Fanuc TP program (LS listing): ultrahose1.ls

/PROG  ultrahose1
/ATTR
COMMENT	= "19-03-19 19:07:18";
PROG_SIZE	= 0;
DEFAULT_GROUP	= 1, *, *, *, *;
/APPL
    ARC Welding Equipment: 1, *, *, *, *;
/MN
   1:  CALL HOME_ALL;
   1:  UFRAME_NUM = 1;
   1:  UTOOL_NUM = 3;
   1:  COL GUARD ADJUST 150;
   1:  PR[91] = PR[90];
   1:  PR[91,1] = PR[90,1] + 11.874;
   1:  PR[91,2] = PR[90,2] + -13.968;
   1:  PR[91,3] = PR[90,3] + 19.695;
   1:  PR[92] = PR[91];
   1:  PR[92,3] = PR[92,3] + 20;
   1:J PR[92] 10% FINE;
   1:L PR[91] R[100]mm/sec CNT100;
   1:  CALL LASER_DRAHT_START;
   1:  PR[91,1] = PR[90,1] + 15.068;
   1:  PR[91,2] = PR[90,2] + -16.411;
   1:L PR[91] R[100]mm/sec CNT100;
   1:  PR[91,1] = PR[90,1] + 15.529;
   1:  PR[91,2] = PR[90,2] + -16.733;
   1:L PR[91] R[100]mm/sec CNT100;
   1:  PR[91,1] = PR[90,1] + 16.034;
   1:  PR[91,2] = PR[90,2] + -16.968;
   1:L PR[91] R[100]mm/sec CNT100;
   1:  PR[91,1] = PR[90,1] + 19.725;
   1:  PR[91,2] = PR[90,2] + -18.490;
   1:L PR[91] R[100]mm/sec CNT100;
   1:  PR[91,1] = PR[90,1] + 20.251;
   1:  PR[91,2] = PR[90,2] + -18.631;
   1:L PR[91] R[100]mm/sec CNT100;
   1:  PR[91,1] = PR[90,1] + 24.153;
   1:  PR[91,2] = PR[90,2] + -19.139;
   1:L PR[91] R[100]mm/sec CNT100;
   1:  PR[91,1] = PR[90,1] + 24.768;
   1:  PR[91,2] = PR[90,2] + -19.192;
   1:L PR[91] R[100]mm/sec CNT100;
   1:  PR[91,1] = PR[90,1] + 25.380;
   1:  PR[91,2] = PR[90,2] + -19.139;
   1:L PR[91] R[100]mm/sec CNT100;
   1:  PR[91,1] = PR[90,1] + 29.249;
   1:  PR[91,2] = PR[90,2] + -18.622;
   1:L PR[91] R[100]mm/sec CNT100;
   1:  PR[91,1] = PR[90,1] + 29.789;
   1:  PR[91,2] = PR[90,2] + -18.477;
   1:L PR[91] R[100]mm/sec CNT100;
   1:  PR[91,1] = PR[90,1] + 30.450;
   1:  PR[91,2] = PR[90,2] + -18.169;
   1:L PR[91] R[100]mm/sec CNT100;
   1:  PR[91,1] = PR[90,1] + 34.024;
   1:  PR[91,2] = PR[90,2] + -16.681;
   1:L PR[91] R[100]mm/sec CNT100;
   1:  PR[91,1] = PR[90,1] + 34.539;
   1:  PR[91,2] = PR[90,2] + -16.320;
   1:L PR[91] R[100]mm/sec CNT100;
   1:  PR[91,1] = PR[90,1] + 37.568;
   1:  PR[91,2] = PR[90,2] + -13.991;
   1:L PR[91] R[100]mm/sec CNT100;
   1:  PR[91,1] = PR[90,1] + 38.026;
   1:  PR[91,2] = PR[90,2] + -13.533;
   1:L PR[91] R[100]mm/sec CNT100;
   1:  PR[91,1] = PR[90,1] + 40.324;
   1:  PR[91,2] = PR[90,2] + -10.530;
   1:L PR[91] R[100]mm/sec CNT100;
   1:  PR[91,1] = PR[90,1] + 40.733;
   1:  PR[91,2] = PR[90,2] + -9.947;
   1:L PR[91] R[100]mm/sec CNT100;
   1:  PR[91,1] = PR[90,1] + 41.032;
   1:  PR[91,2] = PR[90,2] + -9.305;
   1:L PR[91] R[100]mm/sec CNT100;
   1:  PR[91,1] = PR[90,1] + 42.471;
   1:  PR[91,2] = PR[90,2] + -5.824;
   1:L PR[91] R[100]mm/sec CNT100;
   1:  PR[91,1] = PR[90,1] + 42.635;
   1:  PR[91,2] = PR[90,2] + -5.212;
   1:L PR[91] R[100]mm/sec CNT100;
   1:  PR[91,1] = PR[90,1] + 42.704;
   1:  PR[91,2] = PR[90,2] + -4.424;
   1:L PR[91] R[100]mm/sec CNT100;
   1:  PR[91,1] = PR[90,1] + 43.146;
   1:  PR[91,2] = PR[90,2] + -0.638;
   1:L PR[91] R[100]mm/sec CNT100;
   1:  PR[91,1] = PR[90,1] + 43.128;
   1:  PR[91,2] = PR[90,2] + 0.046;
   1:L PR[91] R[100]mm/sec CNT100;
   1:  PR[91,1] = PR[90,1] + 42.647;
   1:  PR[91,2] = PR[90,2] + 3.711;
   1:L PR[91] R[100]mm/sec CNT100;
   1:  PR[91,1] = PR[90,1] + 42.471;
   1:  PR[91,2] = PR[90,2] + 4.366;
   1:L PR[91] R[100]mm/sec CNT100;
   1:  PR[91,1] = PR[90,1] + 41.032;
   1:  PR[91,2] = PR[90,2] + 7.846;
   1:L PR[91] R[100]mm/sec CNT100;
   1:  PR[91,1] = PR[90,1] + 40.733;
   1:  PR[91,2] = PR[90,2] + 8.488;
   1:L PR[91] R[100]mm/sec CNT100;
   1:  PR[91,1] = PR[90,1] + 40.324;
   1:  PR[91,2] = PR[90,2] + 9.072;
   1:L PR[91] R[100]mm/sec CNT100;
   1:  PR[91,1] = PR[90,1] + 38.025;
   1:  PR[91,2] = PR[90,2] + 12.075;
   1:L PR[91] R[100]mm/sec CNT100;
   1:  PR[91,1] = PR[90,1] + 37.567;
   1:  PR[91,2] = PR[90,2] + 12.533;
   1:L PR[91] R[100]mm/sec CNT100;
   1:  PR[91,1] = PR[90,1] + 34.538;
   1:  PR[91,2] = PR[90,2] + 14.862;
   1:L PR[91] R[100]mm/sec CNT100;
   1:  PR[91,1] = PR[90,1] + 33.989;
   1:  PR[91,2] = PR[90,2] + 15.247;
   1:L PR[91] R[100]mm/sec CNT100;
   1:  PR[91,1] = PR[90,1] + 33.379;
   1:  PR[91,2] = PR[90,2] + 15.531;
   1:L PR[91] R[100]mm/sec CNT100;
   1:  PR[91,1] = PR[90,1] + 29.828;
   1:  PR[91,2] = PR[90,2] + 17.008;
   1:L PR[91] R[100]mm/sec CNT100;
   1:  PR[91,1] = PR[90,1] + 29.246;
   1:  PR[91,2] = PR[90,2] + 17.164;
   1:L PR[91] R[100]mm/sec CNT100;
   1:  PR[91,1] = PR[90,1] + 25.377;
   1:  PR[91,2] = PR[90,2] + 17.680;
   1:L PR[91] R[100]mm/sec CNT100;
   1:  PR[91,1] = PR[90,1] + 24.766;
   1:  PR[91,2] = PR[90,2] + 17.734;
   1:L PR[91] R[100]mm/sec CNT100;
   1:  PR[91,1] = PR[90,1] + 24.150;
   1:  PR[91,2] = PR[90,2] + 17.680;
   1:L PR[91] R[100]mm/sec CNT100;
   1:  PR[91,1] = PR[90,1] + 20.249;
   1:  PR[91,2] = PR[90,2] + 17.172;
   1:L PR[91] R[100]mm/sec CNT100;
   1:  PR[91,1] = PR[90,1] + 19.767;
   1:  PR[91,2] = PR[90,2] + 17.043;
   1:L PR[91] R[100]mm/sec CNT100;
   1:  PR[91,1] = PR[90,1] + 19.155;
   1:  PR[91,2] = PR[90,2] + 16.757;
   1:L PR[91] R[100]mm/sec CNT100;
   1:  PR[91,1] = PR[90,1] + 15.490;
   1:  PR[91,2] = PR[90,2] + 15.247;
   1:L PR[91] R[100]mm/sec CNT100;
   1:  PR[91,1] = PR[90,1] + 15.067;
   1:  PR[91,2] = PR[90,2] + 14.951;
   1:L PR[91] R[100]mm/sec CNT100;
   1:  PR[91,1] = PR[90,1] + 11.873;
   1:  PR[91,2] = PR[90,2] + 12.508;
   1:L PR[91] R[100]mm/sec CNT100;
   1:  PR[91,1] = PR[90,1] + 11.527;
   1:  PR[91,2] = PR[90,2] + 12.162;
   1:L PR[91] R[100]mm/sec CNT100;
   1:  PR[91,1] = PR[90,1] + 9.049;
   1:  PR[91,2] = PR[90,2] + 8.939;
   1:L PR[91] R[100]mm/sec CNT100;
   1:  PR[91,1] = PR[90,1] + 8.753;
   1:  PR[91,2] = PR[90,2] + 8.515;
   1:L PR[91] R[100]mm/sec CNT100;
   1:  PR[91,1] = PR[90,1] + 8.534;
   1:  PR[91,2] = PR[90,2] + 8.047;
   1:L PR[91] R[100]mm/sec CNT100;
   1:  PR[91,1] = PR[90,1] + 6.970;
   1:  PR[91,2] = PR[90,2] + 4.277;
   1:L PR[91] R[100]mm/sec CNT100;
   1:  PR[91,1] = PR[90,1] + 6.862;
   1:  PR[91,2] = PR[90,2] + 3.874;
   1:L PR[91] R[100]mm/sec CNT100;
   1:  PR[91,1] = PR[90,1] + 6.811;
   1:  PR[91,2] = PR[90,2] + 3.287;
   1:L PR[91] R[100]mm/sec CNT100;
   1:  PR[91,1] = PR[90,1] + 6.282;
   1:  PR[91,2] = PR[90,2] + -0.772;
   1:L PR[91] R[100]mm/sec CNT100;
   1:  PR[91,1] = PR[90,1] + 6.336;
   1:  PR[91,2] = PR[90,2] + -1.394;
   1:L PR[91] R[100]mm/sec CNT100;
   1:  PR[91,1] = PR[90,1] + 6.851;
   1:  PR[91,2] = PR[90,2] + -5.290;
   1:L PR[91] R[100]mm/sec CNT100;
   1:  PR[91,1] = PR[90,1] + 6.970;
   1:  PR[91,2] = PR[90,2] + -5.736;
   1:L PR[91] R[100]mm/sec CNT100;
   1:  PR[91,1] = PR[90,1] + 8.535;
   1:  PR[91,2] = PR[90,2] + -9.506;
   1:L PR[91] R[100]mm/sec CNT100;
   1:  PR[91,1] = PR[90,1] + 8.753;
   1:  PR[91,2] = PR[90,2] + -9.975;
   1:L PR[91] R[100]mm/sec CNT100;
   1:  PR[91,1] = PR[90,1] + 9.050;
   1:  PR[91,2] = PR[90,2] + -10.398;
   1:L PR[91] R[100]mm/sec CNT100;
   1:  PR[91,1] = PR[90,1] + 11.528;
   1:  PR[91,2] = PR[90,2] + -13.622;
   1:L PR[91] R[100]mm/sec CNT100;
   1:  PR[91,1] = PR[90,1] + 11.874;
   1:  PR[91,2] = PR[90,2] + -13.968;
   1:L PR[91] R[100]mm/sec CNT100TB   .50sec,CALL END_PUD;
   1:  PR[92] = PR[91];
   1:  PR[92,3] = PR[92,3] + 20;
   1:J PR[92] 10% FINE;
   1:  PR[91,1] = PR[90,1] + 59.086;
   1:  PR[91,2] = PR[90,2] + -12.393;
   1:  PR[92] = PR[91];
   1:  PR[92,3] = PR[92,3] + 20;
   1:J PR[92] 10% FINE;
   1:L PR[91] R[100]mm/sec CNT100;
   1:  CALL LASER_DRAHT_START;
   1:  PR[91,1] = PR[90,1] + 60.293;
   1:  PR[91,2] = PR[90,2] + -13.557;
   1:L PR[91] R[100]mm/sec CNT100;
   1:  PR[91,1] = PR[90,1] + 62.143;
   1:  PR[91,2] = PR[90,2] + -15.300;
   1:L PR[91] R[100]mm/sec CNT100;
   1:  PR[91,1] = PR[90,1] + 63.971;
   1:  PR[91,2] = PR[90,2] + -16.401;
   1:L PR[91] R[100]mm/sec CNT100;
   1:  PR[91,1] = PR[90,1] + 65.772;
   1:  PR[91,2] = PR[90,2] + -17.456;
   1:L PR[91] R[100]mm/sec CNT100;
   1:  PR[91,1] = PR[90,1] + 68.248;
   1:  PR[91,2] = PR[90,2] + -18.274;
   1:L PR[91] R[100]mm/sec CNT100;
   1:  PR[91,1] = PR[90,1] + 69.782;
   1:  PR[91,2] = PR[90,2] + -18.759;
   1:L PR[91] R[100]mm/sec CNT100;
   1:  PR[91,1] = PR[90,1] + 72.825;
   1:  PR[91,2] = PR[90,2] + -19.060;
   1:L PR[91] R[100]mm/sec CNT100;
   1:  PR[91,1] = PR[90,1] + 73.969;
   1:  PR[91,2] = PR[90,2] + -19.158;
   1:L PR[91] R[100]mm/sec CNT100;
   1:  PR[91,1] = PR[90,1] + 78.141;
   1:  PR[91,2] = PR[90,2] + -18.634;
   1:L PR[91] R[100]mm/sec CNT100;
   1:  PR[91,1] = PR[90,1] + 81.686;
   1:  PR[91,2] = PR[90,2] + -17.372;
   1:L PR[91] R[100]mm/sec CNT100;
   1:  PR[91,1] = PR[90,1] + 82.061;
   1:  PR[91,2] = PR[90,2] + -17.234;
   1:L PR[91] R[100]mm/sec CNT100;
   1:  PR[91,1] = PR[90,1] + 85.575;
   1:  PR[91,2] = PR[90,2] + -15.011;
   1:L PR[91] R[100]mm/sec CNT100;
   1:  PR[91,1] = PR[90,1] + 88.491;
   1:  PR[91,2] = PR[90,2] + -12.096;
   1:L PR[91] R[100]mm/sec CNT100;
   1:  PR[91,1] = PR[90,1] + 90.677;
   1:  PR[91,2] = PR[90,2] + -8.631;
   1:L PR[91] R[100]mm/sec CNT100;
   1:  PR[91,1] = PR[90,1] + 92.020;
   1:  PR[91,2] = PR[90,2] + -4.770;
   1:L PR[91] R[100]mm/sec CNT100;
   1:  PR[91,1] = PR[90,1] + 92.467;
   1:  PR[91,2] = PR[90,2] + -0.729;
   1:L PR[91] R[100]mm/sec CNT100;
   1:  PR[91,1] = PR[90,1] + 92.020;
   1:  PR[91,2] = PR[90,2] + 3.311;
   1:L PR[91] R[100]mm/sec CNT100;
   1:  PR[91,1] = PR[90,1] + 90.677;
   1:  PR[91,2] = PR[90,2] + 7.172;
   1:L PR[91] R[100]mm/sec CNT100;
   1:  PR[91,1] = PR[90,1] + 88.491;
   1:  PR[91,2] = PR[90,2] + 10.637;
   1:L PR[91] R[100]mm/sec CNT100;
   1:  PR[91,1] = PR[90,1] + 85.575;
   1:  PR[91,2] = PR[90,2] + 13.552;
   1:L PR[91] R[100]mm/sec CNT100;
   1:  PR[91,1] = PR[90,1] + 82.069;
   1:  PR[91,2] = PR[90,2] + 15.770;
   1:L PR[91] R[100]mm/sec CNT100;
   1:  PR[91,1] = PR[90,1] + 78.143;
   1:  PR[91,2] = PR[90,2] + 17.175;
   1:L PR[91] R[100]mm/sec CNT100;
   1:  PR[91,1] = PR[90,1] + 74.809;
   1:  PR[91,2] = PR[90,2] + 17.581;
   1:L PR[91] R[100]mm/sec CNT100;
   1:  PR[91,1] = PR[90,1] + 73.972;
   1:  PR[91,2] = PR[90,2] + 17.696;
   1:L PR[91] R[100]mm/sec CNT100;
   1:  PR[91,1] = PR[90,1] + 70.968;
   1:  PR[91,2] = PR[90,2] + 17.396;
   1:L PR[91] R[100]mm/sec CNT100;
   1:  PR[91,1] = PR[90,1] + 69.783;
   1:  PR[91,2] = PR[90,2] + 17.297;
   1:L PR[91] R[100]mm/sec CNT100;
   1:  PR[91,1] = PR[90,1] + 67.265;
   1:  PR[91,2] = PR[90,2] + 16.462;
   1:L PR[91] R[100]mm/sec CNT100;
   1:  PR[91,1] = PR[90,1] + 65.772;
   1:  PR[91,2] = PR[90,2] + 15.993;
   1:L PR[91] R[100]mm/sec CNT100;
   1:  PR[91,1] = PR[90,1] + 63.838;
   1:  PR[91,2] = PR[90,2] + 14.826;
   1:L PR[91] R[100]mm/sec CNT100;
   1:  PR[91,1] = PR[90,1] + 62.143;
   1:  PR[91,2] = PR[90,2] + 13.837;
   1:L PR[91] R[100]mm/sec CNT100;
   1:  PR[91,1] = PR[90,1] + 60.804;
   1:  PR[91,2] = PR[90,2] + 12.545;
   1:L PR[91] R[100]mm/sec CNT100;
   1:  PR[91,1] = PR[90,1] + 59.084;
   1:  PR[91,2] = PR[90,2] + 10.928;
   1:L PR[91] R[100]mm/sec CNT100;
   1:  PR[91,1] = PR[90,1] + 58.273;
   1:  PR[91,2] = PR[90,2] + 9.680;
   1:L PR[91] R[100]mm/sec CNT100;
   1:  PR[91,1] = PR[90,1] + 56.759;
   1:  PR[91,2] = PR[90,2] + 7.403;
   1:L PR[91] R[100]mm/sec CNT100;
   1:  PR[91,1] = PR[90,1] + 55.312;
   1:  PR[91,2] = PR[90,2] + 3.452;
   1:L PR[91] R[100]mm/sec CNT100;
   1:  PR[91,1] = PR[90,1] + 55.212;
   1:  PR[91,2] = PR[90,2] + 2.599;
   1:L PR[91] R[100]mm/sec CNT100;
   1:  PR[91,1] = PR[90,1] + 55.211;
   1:  PR[91,2] = PR[90,2] + 2.366;
   1:L PR[91] R[100]mm/sec CNT100;
   1:  PR[91,1] = PR[90,1] + 54.847;
   1:  PR[91,2] = PR[90,2] + -0.750;
   1:L PR[91] R[100]mm/sec CNT100;
   1:  PR[91,1] = PR[90,1] + 54.928;
   1:  PR[91,2] = PR[90,2] + -1.594;
   1:L PR[91] R[100]mm/sec CNT100;
   1:  PR[91,1] = PR[90,1] + 55.312;
   1:  PR[91,2] = PR[90,2] + -4.913;
   1:L PR[91] R[100]mm/sec CNT100;
   1:  PR[91,1] = PR[90,1] + 56.761;
   1:  PR[91,2] = PR[90,2] + -8.866;
   1:L PR[91] R[100]mm/sec CNT100;
   1:  PR[91,1] = PR[90,1] + 59.086;
   1:  PR[91,2] = PR[90,2] + -12.393;
   1:L PR[91] R[100]mm/sec CNT100TB   .50sec,CALL END_PUD;
   1:  PR[92] = PR[91];
   1:  PR[92,3] = PR[92,3] + 20;
   1:J PR[92] 10% FINE;
   1:  PR[91,1] = PR[90,1] + -40.837;
   1:  PR[91,2] = PR[90,2] + 7.347;
   1:  PR[92] = PR[91];
   1:  PR[92,3] = PR[92,3] + 20;
   1:J PR[92] 10% FINE;
   1:L PR[91] R[100]mm/sec CNT100;
   1:  CALL LASER_DRAHT_START;
   1:  PR[91,1] = PR[90,1] + -41.039;
   1:  PR[91,2] = PR[90,2] + 6.912;
   1:L PR[91] R[100]mm/sec CNT100;
   1:  PR[91,1] = PR[90,1] + -42.167;
   1:  PR[91,2] = PR[90,2] + 3.679;
   1:L PR[91] R[100]mm/sec CNT100;
   1:  PR[91,1] = PR[90,1] + -42.292;
   1:  PR[91,2] = PR[90,2] + 3.211;
   1:L PR[91] R[100]mm/sec CNT100;
   1:  PR[91,1] = PR[90,1] + -42.343;
   1:  PR[91,2] = PR[90,2] + 2.632;
   1:L PR[91] R[100]mm/sec CNT100;
   1:  PR[91,1] = PR[90,1] + -42.723;
   1:  PR[91,2] = PR[90,2] + -0.754;
   1:L PR[91] R[100]mm/sec CNT100;
   1:  PR[91,1] = PR[90,1] + -42.678;
   1:  PR[91,2] = PR[90,2] + -1.274;
   1:L PR[91] R[100]mm/sec CNT100;
   1:  PR[91,1] = PR[90,1] + -42.298;
   1:  PR[91,2] = PR[90,2] + -4.646;
   1:L PR[91] R[100]mm/sec CNT100;
   1:  PR[91,1] = PR[90,1] + -42.167;
   1:  PR[91,2] = PR[90,2] + -5.137;
   1:L PR[91] R[100]mm/sec CNT100;
   1:  PR[91,1] = PR[90,1] + -41.039;
   1:  PR[91,2] = PR[90,2] + -8.371;
   1:L PR[91] R[100]mm/sec CNT100;
   1:  PR[91,1] = PR[90,1] + -40.837;
   1:  PR[91,2] = PR[90,2] + -8.806;
   1:L PR[91] R[100]mm/sec CNT100;
   1:  PR[91,1] = PR[90,1] + -38.985;
   1:  PR[91,2] = PR[90,2] + -11.762;
   1:L PR[91] R[100]mm/sec CNT100;
   1:  PR[91,1] = PR[90,1] + -38.737;
   1:  PR[91,2] = PR[90,2] + -12.115;
   1:L PR[91] R[100]mm/sec CNT100;
   1:  PR[91,1] = PR[90,1] + -35.914;
   1:  PR[91,2] = PR[90,2] + -14.949;
   1:L PR[91] R[100]mm/sec CNT100;
   1:  PR[91,1] = PR[90,1] + -35.616;
   1:  PR[91,2] = PR[90,2] + -15.158;
   1:L PR[91] R[100]mm/sec CNT100;
   1:  PR[91,1] = PR[90,1] + -32.543;
   1:  PR[91,2] = PR[90,2] + -17.099;
   1:L PR[91] R[100]mm/sec CNT100;
   1:  PR[91,1] = PR[90,1] + -32.290;
   1:  PR[91,2] = PR[90,2] + -17.218;
   1:L PR[91] R[100]mm/sec CNT100;
   1:  PR[91,1] = PR[90,1] + -28.724;
   1:  PR[91,2] = PR[90,2] + -18.475;
   1:L PR[91] R[100]mm/sec CNT100;
   1:  PR[91,1] = PR[90,1] + -28.577;
   1:  PR[91,2] = PR[90,2] + -18.514;
   1:L PR[91] R[100]mm/sec CNT100;
   1:  PR[91,1] = PR[90,1] + -28.319;
   1:  PR[91,2] = PR[90,2] + -18.537;
   1:L PR[91] R[100]mm/sec CNT100;
   1:  PR[91,1] = PR[90,1] + -24.525;
   1:  PR[91,2] = PR[90,2] + -18.980;
   1:L PR[91] R[100]mm/sec CNT100;
   1:  PR[91,1] = PR[90,1] + -20.455;
   1:  PR[91,2] = PR[90,2] + -18.540;
   1:L PR[91] R[100]mm/sec CNT100;
   1:  PR[91,1] = PR[90,1] + -16.577;
   1:  PR[91,2] = PR[90,2] + -17.192;
   1:L PR[91] R[100]mm/sec CNT100;
   1:  PR[91,1] = PR[90,1] + -15.160;
   1:  PR[91,2] = PR[90,2] + -16.307;
   1:L PR[91] R[100]mm/sec CNT100;
   1:  PR[91,1] = PR[90,1] + -13.076;
   1:  PR[91,2] = PR[90,2] + -15.031;
   1:L PR[91] R[100]mm/sec CNT100;
   1:  PR[91,1] = PR[90,1] + -10.125;
   1:  PR[91,2] = PR[90,2] + -12.150;
   1:L PR[91] R[100]mm/sec CNT100;
   1:  PR[91,1] = PR[90,1] + -7.899;
   1:  PR[91,2] = PR[90,2] + -8.685;
   1:L PR[91] R[100]mm/sec CNT100;
   1:  PR[91,1] = PR[90,1] + -6.516;
   1:  PR[91,2] = PR[90,2] + -4.813;
   1:L PR[91] R[100]mm/sec CNT100;
   1:  PR[91,1] = PR[90,1] + -6.050;
   1:  PR[91,2] = PR[90,2] + -0.729;
   1:L PR[91] R[100]mm/sec CNT100;
   1:  PR[91,1] = PR[90,1] + -6.492;
   1:  PR[91,2] = PR[90,2] + 3.146;
   1:L PR[91] R[100]mm/sec CNT100;
   1:  PR[91,1] = PR[90,1] + -6.516;
   1:  PR[91,2] = PR[90,2] + 3.353;
   1:L PR[91] R[100]mm/sec CNT100;
   1:  PR[91,1] = PR[90,1] + -7.899;
   1:  PR[91,2] = PR[90,2] + 7.226;
   1:L PR[91] R[100]mm/sec CNT100;
   1:  PR[91,1] = PR[90,1] + -10.125;
   1:  PR[91,2] = PR[90,2] + 10.691;
   1:L PR[91] R[100]mm/sec CNT100;
   1:  PR[91,1] = PR[90,1] + -13.076;
   1:  PR[91,2] = PR[90,2] + 13.573;
   1:L PR[91] R[100]mm/sec CNT100;
   1:  PR[91,1] = PR[90,1] + -15.160;
   1:  PR[91,2] = PR[90,2] + 14.848;
   1:L PR[91] R[100]mm/sec CNT100;
   1:  PR[91,1] = PR[90,1] + -16.577;
   1:  PR[91,2] = PR[90,2] + 15.733;
   1:L PR[91] R[100]mm/sec CNT100;
   1:  PR[91,1] = PR[90,1] + -20.455;
   1:  PR[91,2] = PR[90,2] + 17.081;
   1:L PR[91] R[100]mm/sec CNT100;
   1:  PR[91,1] = PR[90,1] + -24.527;
   1:  PR[91,2] = PR[90,2] + 17.522;
   1:L PR[91] R[100]mm/sec CNT100;
   1:  PR[91,1] = PR[90,1] + -28.551;
   1:  PR[91,2] = PR[90,2] + 17.062;
   1:L PR[91] R[100]mm/sec CNT100;
   1:  PR[91,1] = PR[90,1] + -28.724;
   1:  PR[91,2] = PR[90,2] + 17.016;
   1:L PR[91] R[100]mm/sec CNT100;
   1:  PR[91,1] = PR[90,1] + -32.290;
   1:  PR[91,2] = PR[90,2] + 15.759;
   1:L PR[91] R[100]mm/sec CNT100;
   1:  PR[91,1] = PR[90,1] + -32.543;
   1:  PR[91,2] = PR[90,2] + 15.640;
   1:L PR[91] R[100]mm/sec CNT100;
   1:  PR[91,1] = PR[90,1] + -35.616;
   1:  PR[91,2] = PR[90,2] + 13.699;
   1:L PR[91] R[100]mm/sec CNT100;
   1:  PR[91,1] = PR[90,1] + -35.914;
   1:  PR[91,2] = PR[90,2] + 13.490;
   1:L PR[91] R[100]mm/sec CNT100;
   1:  PR[91,1] = PR[90,1] + -38.737;
   1:  PR[91,2] = PR[90,2] + 10.656;
   1:L PR[91] R[100]mm/sec CNT100;
   1:  PR[91,1] = PR[90,1] + -38.984;
   1:  PR[91,2] = PR[90,2] + 10.303;
   1:L PR[91] R[100]mm/sec CNT100;
   1:  PR[91,1] = PR[90,1] + -40.837;
   1:  PR[91,2] = PR[90,2] + 7.347;
   1:L PR[91] R[100]mm/sec CNT100TB   .50sec,CALL END_PUD;
   1:  PR[92] = PR[91];
   1:  PR[92,3] = PR[92,3] + 20;
   1:J PR[92] 10% FINE;
   1:  PR[91,1] = PR[90,1] + -83.415;
   1:  PR[91,2] = PR[90,2] + 14.998;
   1:  PR[92] = PR[91];
   1:  PR[92,3] = PR[92,3] + 20;
   1:J PR[92] 10% FINE;
   1:L PR[91] R[100]mm/sec CNT100;
   1:  CALL LASER_DRAHT_START;
   1:  PR[91,1] = PR[90,1] + -86.519;
   1:  PR[91,2] = PR[90,2] + 12.750;
   1:L PR[91] R[100]mm/sec CNT100;
   1:  PR[91,1] = PR[90,1] + -89.079;
   1:  PR[91,2] = PR[90,2] + 9.920;
   1:L PR[91] R[100]mm/sec CNT100;
   1:  PR[91,1] = PR[90,1] + -90.989;
   1:  PR[91,2] = PR[90,2] + 6.634;
   1:L PR[91] R[100]mm/sec CNT100;
   1:  PR[91,1] = PR[90,1] + -92.167;
   1:  PR[91,2] = PR[90,2] + 3.033;
   1:L PR[91] R[100]mm/sec CNT100;
   1:  PR[91,1] = PR[90,1] + -92.552;
   1:  PR[91,2] = PR[90,2] + -0.594;
   1:L PR[91] R[100]mm/sec CNT100;
   1:  PR[91,1] = PR[90,1] + -92.516;
   1:  PR[91,2] = PR[90,2] + -0.742;
   1:L PR[91] R[100]mm/sec CNT100;
   1:  PR[91,1] = PR[90,1] + -92.124;
   1:  PR[91,2] = PR[90,2] + -4.484;
   1:L PR[91] R[100]mm/sec CNT100;
   1:  PR[91,1] = PR[90,1] + -92.092;
   1:  PR[91,2] = PR[90,2] + -4.604;
   1:L PR[91] R[100]mm/sec CNT100;
   1:  PR[91,1] = PR[90,1] + -90.966;
   1:  PR[91,2] = PR[90,2] + -8.078;
   1:L PR[91] R[100]mm/sec CNT100;
   1:  PR[91,1] = PR[90,1] + -90.932;
   1:  PR[91,2] = PR[90,2] + -8.151;
   1:L PR[91] R[100]mm/sec CNT100;
   1:  PR[91,1] = PR[90,1] + -89.070;
   1:  PR[91,2] = PR[90,2] + -11.382;
   1:L PR[91] R[100]mm/sec CNT100;
   1:  PR[91,1] = PR[90,1] + -89.064;
   1:  PR[91,2] = PR[90,2] + -11.391;
   1:L PR[91] R[100]mm/sec CNT100;
   1:  PR[91,1] = PR[90,1] + -86.510;
   1:  PR[91,2] = PR[90,2] + -14.226;
   1:L PR[91] R[100]mm/sec CNT100;
   1:  PR[91,1] = PR[90,1] + -83.462;
   1:  PR[91,2] = PR[90,2] + -16.448;
   1:L PR[91] R[100]mm/sec CNT100;
   1:  PR[91,1] = PR[90,1] + -79.943;
   1:  PR[91,2] = PR[90,2] + -18.018;
   1:L PR[91] R[100]mm/sec CNT100;
   1:  PR[91,1] = PR[90,1] + -76.158;
   1:  PR[91,2] = PR[90,2] + -18.839;
   1:L PR[91] R[100]mm/sec CNT100;
   1:  PR[91,1] = PR[90,1] + -72.275;
   1:  PR[91,2] = PR[90,2] + -18.873;
   1:L PR[91] R[100]mm/sec CNT100;
   1:  PR[91,1] = PR[90,1] + -68.461;
   1:  PR[91,2] = PR[90,2] + -18.113;
   1:L PR[91] R[100]mm/sec CNT100;
   1:  PR[91,1] = PR[90,1] + -64.885;
   1:  PR[91,2] = PR[90,2] + -16.588;
   1:L PR[91] R[100]mm/sec CNT100;
   1:  PR[91,1] = PR[90,1] + -61.704;
   1:  PR[91,2] = PR[90,2] + -14.363;
   1:L PR[91] R[100]mm/sec CNT100;
   1:  PR[91,1] = PR[90,1] + -59.064;
   1:  PR[91,2] = PR[90,2] + -11.529;
   1:L PR[91] R[100]mm/sec CNT100;
   1:  PR[91,1] = PR[90,1] + -57.083;
   1:  PR[91,2] = PR[90,2] + -8.212;
   1:L PR[91] R[100]mm/sec CNT100;
   1:  PR[91,1] = PR[90,1] + -55.857;
   1:  PR[91,2] = PR[90,2] + -4.558;
   1:L PR[91] R[100]mm/sec CNT100;
   1:  PR[91,1] = PR[90,1] + -55.668;
   1:  PR[91,2] = PR[90,2] + -2.815;
   1:L PR[91] R[100]mm/sec CNT100;
   1:  PR[91,1] = PR[90,1] + -55.618;
   1:  PR[91,2] = PR[90,2] + -1.089;
   1:L PR[91] R[100]mm/sec CNT100;
   1:  PR[91,1] = PR[90,1] + -55.578;
   1:  PR[91,2] = PR[90,2] + -0.668;
   1:L PR[91] R[100]mm/sec CNT100;
   1:  PR[91,1] = PR[90,1] + -55.613;
   1:  PR[91,2] = PR[90,2] + 0.420;
   1:L PR[91] R[100]mm/sec CNT100;
   1:  PR[91,1] = PR[90,1] + -55.902;
   1:  PR[91,2] = PR[90,2] + 3.098;
   1:L PR[91] R[100]mm/sec CNT100;
   1:  PR[91,1] = PR[90,1] + -57.123;
   1:  PR[91,2] = PR[90,2] + 6.752;
   1:L PR[91] R[100]mm/sec CNT100;
   1:  PR[91,1] = PR[90,1] + -59.096;
   1:  PR[91,2] = PR[90,2] + 10.069;
   1:L PR[91] R[100]mm/sec CNT100;
   1:  PR[91,1] = PR[90,1] + -61.725;
   1:  PR[91,2] = PR[90,2] + 12.904;
   1:L PR[91] R[100]mm/sec CNT100;
   1:  PR[91,1] = PR[90,1] + -64.896;
   1:  PR[91,2] = PR[90,2] + 15.132;
   1:L PR[91] R[100]mm/sec CNT100;
   1:  PR[91,1] = PR[90,1] + -67.021;
   1:  PR[91,2] = PR[90,2] + 16.050;
   1:L PR[91] R[100]mm/sec CNT100;
   1:  PR[91,1] = PR[90,1] + -68.452;
   1:  PR[91,2] = PR[90,2] + 16.656;
   1:L PR[91] R[100]mm/sec CNT100;
   1:  PR[91,1] = PR[90,1] + -72.257;
   1:  PR[91,2] = PR[90,2] + 17.419;
   1:L PR[91] R[100]mm/sec CNT100;
   1:  PR[91,1] = PR[90,1] + -76.127;
   1:  PR[91,2] = PR[90,2] + 17.388;
   1:L PR[91] R[100]mm/sec CNT100;
   1:  PR[91,1] = PR[90,1] + -79.901;
   1:  PR[91,2] = PR[90,2] + 16.568;
   1:L PR[91] R[100]mm/sec CNT100;
   1:  PR[91,1] = PR[90,1] + -83.415;
   1:  PR[91,2] = PR[90,2] + 14.998;
   1:L PR[91] R[100]mm/sec CNT100TB   .50sec,CALL END_PUD;
   1:  PR[92] = PR[91];
   1:  PR[92,3] = PR[92,3] + 20;
   1:J PR[92] 10% FINE;
   1:  PR[91] = PR[90];
   1:  PR[91,1] = PR[90,1] + 80.831;
   1:  PR[91,2] = PR[90,2] + -17.694;
   1:  PR[91,3] = PR[90,3] + 20.995;
   1:  PR[92] = PR[91];
   1:  PR[92,3] = PR[92,3] + 20;
   1:J PR[92] 10% FINE;
   1:L PR[91] R[100]mm/sec CNT100;
   1:  CALL LASER_DRAHT_START;
   1:  PR[91,1] = PR[90,1] + 81.864;
   1:  PR[91,2] = PR[90,2] + -17.313;
   1:L PR[91] R[100]mm/sec CNT100;
   1:  PR[91,1] = PR[90,1] + 85.391;
   1:  PR[91,2] = PR[90,2] + -15.076;
   1:L PR[91] R[100]mm/sec CNT100;
   1:  PR[91,1] = PR[90,1] + 88.316;
   1:  PR[91,2] = PR[90,2] + -12.145;
   1:L PR[91] R[100]mm/sec CNT100;
   1:  PR[91,1] = PR[90,1] + 90.510;
   1:  PR[91,2] = PR[90,2] + -8.661;
   1:L PR[91] R[100]mm/sec CNT100;
   1:  PR[91,1] = PR[90,1] + 91.869;
   1:  PR[91,2] = PR[90,2] + -4.791;
   1:L PR[91] R[100]mm/sec CNT100;
   1:  PR[91,1] = PR[90,1] + 92.323;
   1:  PR[91,2] = PR[90,2] + -0.849;
   1:L PR[91] R[100]mm/sec CNT100;
   1:  PR[91,1] = PR[90,1] + 92.347;
   1:  PR[91,2] = PR[90,2] + -0.692;
   1:L PR[91] R[100]mm/sec CNT100;
   1:  PR[91,1] = PR[90,1] + 91.953;
   1:  PR[91,2] = PR[90,2] + 2.747;
   1:L PR[91] R[100]mm/sec CNT100;
   1:  PR[91,1] = PR[90,1] + 91.901;
   1:  PR[91,2] = PR[90,2] + 3.027;
   1:L PR[91] R[100]mm/sec CNT100;
   1:  PR[91,1] = PR[90,1] + 91.867;
   1:  PR[91,2] = PR[90,2] + 3.336;
   1:L PR[91] R[100]mm/sec CNT100;
   1:  PR[91,1] = PR[90,1] + 90.510;
   1:  PR[91,2] = PR[90,2] + 7.202;
   1:L PR[91] R[100]mm/sec CNT100;
   1:  PR[91,1] = PR[90,1] + 88.316;
   1:  PR[91,2] = PR[90,2] + 10.686;
   1:L PR[91] R[100]mm/sec CNT100;
   1:  PR[91,1] = PR[90,1] + 85.391;
   1:  PR[91,2] = PR[90,2] + 13.617;
   1:L PR[91] R[100]mm/sec CNT100;
   1:  PR[91,1] = PR[90,1] + 81.874;
   1:  PR[91,2] = PR[90,2] + 15.848;
   1:L PR[91] R[100]mm/sec CNT100;
   1:  PR[91,1] = PR[90,1] + 78.992;
   1:  PR[91,2] = PR[90,2] + 16.872;
   1:L PR[91] R[100]mm/sec CNT100;
   1:  PR[91,1] = PR[90,1] + 77.920;
   1:  PR[91,2] = PR[90,2] + 17.269;
   1:L PR[91] R[100]mm/sec CNT100;
   1:  PR[91,1] = PR[90,1] + 75.202;
   1:  PR[91,2] = PR[90,2] + 17.601;
   1:L PR[91] R[100]mm/sec CNT100;
   1:  PR[91,1] = PR[90,1] + 73.738;
   1:  PR[91,2] = PR[90,2] + 17.801;
   1:L PR[91] R[100]mm/sec CNT100;
   1:  PR[91,1] = PR[90,1] + 71.378;
   1:  PR[91,2] = PR[90,2] + 17.566;
   1:L PR[91] R[100]mm/sec CNT100;
   1:  PR[91,1] = PR[90,1] + 69.523;
   1:  PR[91,2] = PR[90,2] + 17.410;
   1:L PR[91] R[100]mm/sec CNT100;
   1:  PR[91,1] = PR[90,1] + 67.660;
   1:  PR[91,2] = PR[90,2] + 16.793;
   1:L PR[91] R[100]mm/sec CNT100;
   1:  PR[91,1] = PR[90,1] + 65.482;
   1:  PR[91,2] = PR[90,2] + 16.108;
   1:L PR[91] R[100]mm/sec CNT100;
   1:  PR[91,1] = PR[90,1] + 64.181;
   1:  PR[91,2] = PR[90,2] + 15.323;
   1:L PR[91] R[100]mm/sec CNT100;
   1:  PR[91,1] = PR[90,1] + 61.820;
   1:  PR[91,2] = PR[90,2] + 13.947;
   1:L PR[91] R[100]mm/sec CNT100;
   1:  PR[91,1] = PR[90,1] + 61.052;
   1:  PR[91,2] = PR[90,2] + 13.205;
   1:L PR[91] R[100]mm/sec CNT100;
   1:  PR[91,1] = PR[90,1] + 58.723;
   1:  PR[91,2] = PR[90,2] + 11.017;
   1:L PR[91] R[100]mm/sec CNT100;
   1:  PR[91,1] = PR[90,1] + 56.378;
   1:  PR[91,2] = PR[90,2] + 7.474;
   1:L PR[91] R[100]mm/sec CNT100;
   1:  PR[91,1] = PR[90,1] + 54.912;
   1:  PR[91,2] = PR[90,2] + 3.488;
   1:L PR[91] R[100]mm/sec CNT100;
   1:  PR[91,1] = PR[90,1] + 54.908;
   1:  PR[91,2] = PR[90,2] + 3.454;
   1:L PR[91] R[100]mm/sec CNT100;
   1:  PR[91,1] = PR[90,1] + 54.425;
   1:  PR[91,2] = PR[90,2] + -0.729;
   1:L PR[91] R[100]mm/sec CNT100;
   1:  PR[91,1] = PR[90,1] + 54.912;
   1:  PR[91,2] = PR[90,2] + -4.949;
   1:L PR[91] R[100]mm/sec CNT100;
   1:  PR[91,1] = PR[90,1] + 56.378;
   1:  PR[91,2] = PR[90,2] + -8.933;
   1:L PR[91] R[100]mm/sec CNT100;
   1:  PR[91,1] = PR[90,1] + 58.730;
   1:  PR[91,2] = PR[90,2] + -12.487;
   1:L PR[91] R[100]mm/sec CNT100;
   1:  PR[91,1] = PR[90,1] + 59.261;
   1:  PR[91,2] = PR[90,2] + -12.998;
   1:L PR[91] R[100]mm/sec CNT100;
   1:  PR[91,1] = PR[90,1] + 61.820;
   1:  PR[91,2] = PR[90,2] + -15.409;
   1:L PR[91] R[100]mm/sec CNT100;
   1:  PR[91,1] = PR[90,1] + 62.881;
   1:  PR[91,2] = PR[90,2] + -16.048;
   1:L PR[91] R[100]mm/sec CNT100;
   1:  PR[91,1] = PR[90,1] + 65.482;
   1:  PR[91,2] = PR[90,2] + -17.571;
   1:L PR[91] R[100]mm/sec CNT100;
   1:  PR[91,1] = PR[90,1] + 67.157;
   1:  PR[91,2] = PR[90,2] + -18.125;
   1:L PR[91] R[100]mm/sec CNT100;
   1:  PR[91,1] = PR[90,1] + 69.522;
   1:  PR[91,2] = PR[90,2] + -18.872;
   1:L PR[91] R[100]mm/sec CNT100;
   1:  PR[91,1] = PR[90,1] + 71.781;
   1:  PR[91,2] = PR[90,2] + -19.095;
   1:L PR[91] R[100]mm/sec CNT100;
   1:  PR[91,1] = PR[90,1] + 73.738;
   1:  PR[91,2] = PR[90,2] + -19.263;
   1:L PR[91] R[100]mm/sec CNT100;
   1:  PR[91,1] = PR[90,1] + 76.433;
   1:  PR[91,2] = PR[90,2] + -18.932;
   1:L PR[91] R[100]mm/sec CNT100;
   1:  PR[91,1] = PR[90,1] + 77.920;
   1:  PR[91,2] = PR[90,2] + -18.731;
   1:L PR[91] R[100]mm/sec CNT100;
   1:  PR[91,1] = PR[90,1] + 80.831;
   1:  PR[91,2] = PR[90,2] + -17.694;
   1:L PR[91] R[100]mm/sec CNT100TB   .50sec,CALL END_PUD;
   1:  PR[92] = PR[91];
   1:  PR[92,3] = PR[92,3] + 20;
   1:J PR[92] 10% FINE;
   1:  PR[91,1] = PR[90,1] + 24.442;
   1:  PR[91,2] = PR[90,2] + 17.762;
   1:  PR[92] = PR[91];
   1:  PR[92,3] = PR[92,3] + 20;
   1:J PR[92] 10% FINE;
   1:L PR[91] R[100]mm/sec CNT100;
   1:  CALL LASER_DRAHT_START;
   1:  PR[91,1] = PR[90,1] + 20.061;
   1:  PR[91,2] = PR[90,2] + 17.192;
   1:L PR[91] R[100]mm/sec CNT100;
   1:  PR[91,1] = PR[90,1] + 19.885;
   1:  PR[91,2] = PR[90,2] + 17.145;
   1:L PR[91] R[100]mm/sec CNT100;
   1:  PR[91,1] = PR[90,1] + 19.558;
   1:  PR[91,2] = PR[90,2] + 16.993;
   1:L PR[91] R[100]mm/sec CNT100;
   1:  PR[91,1] = PR[90,1] + 15.442;
   1:  PR[91,2] = PR[90,2] + 15.297;
   1:L PR[91] R[100]mm/sec CNT100;
   1:  PR[91,1] = PR[90,1] + 15.281;
   1:  PR[91,2] = PR[90,2] + 15.184;
   1:L PR[91] R[100]mm/sec CNT100;
   1:  PR[91,1] = PR[90,1] + 11.695;
   1:  PR[91,2] = PR[90,2] + 12.441;
   1:L PR[91] R[100]mm/sec CNT100;
   1:  PR[91,1] = PR[90,1] + 11.575;
   1:  PR[91,2] = PR[90,2] + 12.322;
   1:L PR[91] R[100]mm/sec CNT100;
   1:  PR[91,1] = PR[90,1] + 8.793;
   1:  PR[91,2] = PR[90,2] + 8.703;
   1:L PR[91] R[100]mm/sec CNT100;
   1:  PR[91,1] = PR[90,1] + 8.683;
   1:  PR[91,2] = PR[90,2] + 8.545;
   1:L PR[91] R[100]mm/sec CNT100;
   1:  PR[91,1] = PR[90,1] + 8.601;
   1:  PR[91,2] = PR[90,2] + 8.370;
   1:L PR[91] R[100]mm/sec CNT100;
   1:  PR[91,1] = PR[90,1] + 6.845;
   1:  PR[91,2] = PR[90,2] + 4.137;
   1:L PR[91] R[100]mm/sec CNT100;
   1:  PR[91,1] = PR[90,1] + 6.821;
   1:  PR[91,2] = PR[90,2] + 4.049;
   1:L PR[91] R[100]mm/sec CNT100;
   1:  PR[91,1] = PR[90,1] + 6.798;
   1:  PR[91,2] = PR[90,2] + 3.785;
   1:L PR[91] R[100]mm/sec CNT100;
   1:  PR[91,1] = PR[90,1] + 6.205;
   1:  PR[91,2] = PR[90,2] + -0.772;
   1:L PR[91] R[100]mm/sec CNT100;
   1:  PR[91,1] = PR[90,1] + 6.232;
   1:  PR[91,2] = PR[90,2] + -1.090;
   1:L PR[91] R[100]mm/sec CNT100;
   1:  PR[91,1] = PR[90,1] + 6.810;
   1:  PR[91,2] = PR[90,2] + -5.465;
   1:L PR[91] R[100]mm/sec CNT100;
   1:  PR[91,1] = PR[90,1] + 6.845;
   1:  PR[91,2] = PR[90,2] + -5.596;
   1:L PR[91] R[100]mm/sec CNT100;
   1:  PR[91,1] = PR[90,1] + 8.601;
   1:  PR[91,2] = PR[90,2] + -9.829;
   1:L PR[91] R[100]mm/sec CNT100;
   1:  PR[91,1] = PR[90,1] + 8.683;
   1:  PR[91,2] = PR[90,2] + -10.004;
   1:L PR[91] R[100]mm/sec CNT100;
   1:  PR[91,1] = PR[90,1] + 8.794;
   1:  PR[91,2] = PR[90,2] + -10.162;
   1:L PR[91] R[100]mm/sec CNT100;
   1:  PR[91,1] = PR[90,1] + 11.576;
   1:  PR[91,2] = PR[90,2] + -13.781;
   1:L PR[91] R[100]mm/sec CNT100;
   1:  PR[91,1] = PR[90,1] + 11.695;
   1:  PR[91,2] = PR[90,2] + -13.900;
   1:L PR[91] R[100]mm/sec CNT100;
   1:  PR[91,1] = PR[90,1] + 15.281;
   1:  PR[91,2] = PR[90,2] + -16.643;
   1:L PR[91] R[100]mm/sec CNT100;
   1:  PR[91,1] = PR[90,1] + 15.480;
   1:  PR[91,2] = PR[90,2] + -16.782;
   1:L PR[91] R[100]mm/sec CNT100;
   1:  PR[91,1] = PR[90,1] + 15.697;
   1:  PR[91,2] = PR[90,2] + -16.883;
   1:L PR[91] R[100]mm/sec CNT100;
   1:  PR[91,1] = PR[90,1] + 19.842;
   1:  PR[91,2] = PR[90,2] + -18.592;
   1:L PR[91] R[100]mm/sec CNT100;
   1:  PR[91,1] = PR[90,1] + 20.063;
   1:  PR[91,2] = PR[90,2] + -18.651;
   1:L PR[91] R[100]mm/sec CNT100;
   1:  PR[91,1] = PR[90,1] + 24.444;
   1:  PR[91,2] = PR[90,2] + -19.221;
   1:L PR[91] R[100]mm/sec CNT100;
   1:  PR[91,1] = PR[90,1] + 24.748;
   1:  PR[91,2] = PR[90,2] + -19.248;
   1:L PR[91] R[100]mm/sec CNT100;
   1:  PR[91,1] = PR[90,1] + 25.049;
   1:  PR[91,2] = PR[90,2] + -19.221;
   1:L PR[91] R[100]mm/sec CNT100;
   1:  PR[91,1] = PR[90,1] + 29.394;
   1:  PR[91,2] = PR[90,2] + -18.641;
   1:L PR[91] R[100]mm/sec CNT100;
   1:  PR[91,1] = PR[90,1] + 29.636;
   1:  PR[91,2] = PR[90,2] + -18.576;
   1:L PR[91] R[100]mm/sec CNT100;
   1:  PR[91,1] = PR[90,1] + 30.018;
   1:  PR[91,2] = PR[90,2] + -18.398;
   1:L PR[91] R[100]mm/sec CNT100;
   1:  PR[91,1] = PR[90,1] + 34.032;
   1:  PR[91,2] = PR[90,2] + -16.727;
   1:L PR[91] R[100]mm/sec CNT100;
   1:  PR[91,1] = PR[90,1] + 34.296;
   1:  PR[91,2] = PR[90,2] + -16.542;
   1:L PR[91] R[100]mm/sec CNT100;
   1:  PR[91,1] = PR[90,1] + 37.698;
   1:  PR[91,2] = PR[90,2] + -13.926;
   1:L PR[91] R[100]mm/sec CNT100;
   1:  PR[91,1] = PR[90,1] + 37.942;
   1:  PR[91,2] = PR[90,2] + -13.682;
   1:L PR[91] R[100]mm/sec CNT100;
   1:  PR[91,1] = PR[90,1] + 40.523;
   1:  PR[91,2] = PR[90,2] + -10.309;
   1:L PR[91] R[100]mm/sec CNT100;
   1:  PR[91,1] = PR[90,1] + 40.759;
   1:  PR[91,2] = PR[90,2] + -9.973;
   1:L PR[91] R[100]mm/sec CNT100;
   1:  PR[91,1] = PR[90,1] + 40.931;
   1:  PR[91,2] = PR[90,2] + -9.604;
   1:L PR[91] R[100]mm/sec CNT100;
   1:  PR[91,1] = PR[90,1] + 42.547;
   1:  PR[91,2] = PR[90,2] + -5.695;
   1:L PR[91] R[100]mm/sec CNT100;
   1:  PR[91,1] = PR[90,1] + 42.634;
   1:  PR[91,2] = PR[90,2] + -5.372;
   1:L PR[91] R[100]mm/sec CNT100;
   1:  PR[91,1] = PR[90,1] + 42.676;
   1:  PR[91,2] = PR[90,2] + -4.882;
   1:L PR[91] R[100]mm/sec CNT100;
   1:  PR[91,1] = PR[90,1] + 43.043;
   1:  PR[91,2] = PR[90,2] + -1.743;
   1:L PR[91] R[100]mm/sec CNT100;
   1:  PR[91,1] = PR[90,1] + 43.191;
   1:  PR[91,2] = PR[90,2] + -0.613;
   1:L PR[91] R[100]mm/sec CNT100;
   1:  PR[91,1] = PR[90,1] + 43.186;
   1:  PR[91,2] = PR[90,2] + -0.242;
   1:L PR[91] R[100]mm/sec CNT100;
   1:  PR[91,1] = PR[90,1] + 42.645;
   1:  PR[91,2] = PR[90,2] + 3.871;
   1:L PR[91] R[100]mm/sec CNT100;
   1:  PR[91,1] = PR[90,1] + 42.547;
   1:  PR[91,2] = PR[90,2] + 4.236;
   1:L PR[91] R[100]mm/sec CNT100;
   1:  PR[91,1] = PR[90,1] + 40.931;
   1:  PR[91,2] = PR[90,2] + 8.145;
   1:L PR[91] R[100]mm/sec CNT100;
   1:  PR[91,1] = PR[90,1] + 40.759;
   1:  PR[91,2] = PR[90,2] + 8.514;
   1:L PR[91] R[100]mm/sec CNT100;
   1:  PR[91,1] = PR[90,1] + 40.523;
   1:  PR[91,2] = PR[90,2] + 8.851;
   1:L PR[91] R[100]mm/sec CNT100;
   1:  PR[91,1] = PR[90,1] + 37.942;
   1:  PR[91,2] = PR[90,2] + 12.223;
   1:L PR[91] R[100]mm/sec CNT100;
   1:  PR[91,1] = PR[90,1] + 37.697;
   1:  PR[91,2] = PR[90,2] + 12.467;
   1:L PR[91] R[100]mm/sec CNT100;
   1:  PR[91,1] = PR[90,1] + 34.296;
   1:  PR[91,2] = PR[90,2] + 15.084;
   1:L PR[91] R[100]mm/sec CNT100;
   1:  PR[91,1] = PR[90,1] + 33.997;
   1:  PR[91,2] = PR[90,2] + 15.293;
   1:L PR[91] R[100]mm/sec CNT100;
   1:  PR[91,1] = PR[90,1] + 33.665;
   1:  PR[91,2] = PR[90,2] + 15.447;
   1:L PR[91] R[100]mm/sec CNT100;
   1:  PR[91,1] = PR[90,1] + 29.676;
   1:  PR[91,2] = PR[90,2] + 17.107;
   1:L PR[91] R[100]mm/sec CNT100;
   1:  PR[91,1] = PR[90,1] + 29.393;
   1:  PR[91,2] = PR[90,2] + 17.183;
   1:L PR[91] R[100]mm/sec CNT100;
   1:  PR[91,1] = PR[90,1] + 25.048;
   1:  PR[91,2] = PR[90,2] + 17.763;
   1:L PR[91] R[100]mm/sec CNT100;
   1:  PR[91,1] = PR[90,1] + 24.747;
   1:  PR[91,2] = PR[90,2] + 17.789;
   1:L PR[91] R[100]mm/sec CNT100;
   1:  PR[91,1] = PR[90,1] + 24.442;
   1:  PR[91,2] = PR[90,2] + 17.762;
   1:L PR[91] R[100]mm/sec CNT100TB   .50sec,CALL END_PUD;
   1:  PR[92] = PR[91];
   1:  PR[92,3] = PR[92,3] + 20;
   1:J PR[92] 10% FINE;
   1:  PR[91,1] = PR[90,1] + -6.135;
   1:  PR[91,2] = PR[90,2] + 2.613;
   1:  PR[92] = PR[91];
   1:  PR[92,3] = PR[92,3] + 20;
   1:J PR[92] 10% FINE;
   1:L PR[91] R[100]mm/sec CNT100;
   1:  CALL LASER_DRAHT_START;
   1:  PR[91,1] = PR[90,1] + -6.132;
   1:  PR[91,2] = PR[90,2] + 2.696;
   1:L PR[91] R[100]mm/sec CNT100;
   1:  PR[91,1] = PR[90,1] + -6.211;
   1:  PR[91,2] = PR[90,2] + 3.378;
   1:L PR[91] R[100]mm/sec CNT100;
   1:  PR[91,1] = PR[90,1] + -7.605;
   1:  PR[91,2] = PR[90,2] + 7.273;
   1:L PR[91] R[100]mm/sec CNT100;
   1:  PR[91,1] = PR[90,1] + -9.848;
   1:  PR[91,2] = PR[90,2] + 10.758;
   1:L PR[91] R[100]mm/sec CNT100;
   1:  PR[91,1] = PR[90,1] + -12.457;
   1:  PR[91,2] = PR[90,2] + 13.307;
   1:L PR[91] R[100]mm/sec CNT100;
   1:  PR[91,1] = PR[90,1] + -12.812;
   1:  PR[91,2] = PR[90,2] + 13.649;
   1:L PR[91] R[100]mm/sec CNT100;
   1:  PR[91,1] = PR[90,1] + -16.362;
   1:  PR[91,2] = PR[90,2] + 15.815;
   1:L PR[91] R[100]mm/sec CNT100;
   1:  PR[91,1] = PR[90,1] + -20.298;
   1:  PR[91,2] = PR[90,2] + 17.139;
   1:L PR[91] R[100]mm/sec CNT100;
   1:  PR[91,1] = PR[90,1] + -24.426;
   1:  PR[91,2] = PR[90,2] + 17.565;
   1:L PR[91] R[100]mm/sec CNT100;
   1:  PR[91,1] = PR[90,1] + -28.515;
   1:  PR[91,2] = PR[90,2] + 17.080;
   1:L PR[91] R[100]mm/sec CNT100;
   1:  PR[91,1] = PR[90,1] + -32.385;
   1:  PR[91,2] = PR[90,2] + 15.719;
   1:L PR[91] R[100]mm/sec CNT100;
   1:  PR[91,1] = PR[90,1] + -35.811;
   1:  PR[91,2] = PR[90,2] + 13.555;
   1:L PR[91] R[100]mm/sec CNT100;
   1:  PR[91,1] = PR[90,1] + -35.829;
   1:  PR[91,2] = PR[90,2] + 13.542;
   1:L PR[91] R[100]mm/sec CNT100;
   1:  PR[91,1] = PR[90,1] + -38.724;
   1:  PR[91,2] = PR[90,2] + 10.635;
   1:L PR[91] R[100]mm/sec CNT100;
   1:  PR[91,1] = PR[90,1] + -38.780;
   1:  PR[91,2] = PR[90,2] + 10.555;
   1:L PR[91] R[100]mm/sec CNT100;
   1:  PR[91,1] = PR[90,1] + -40.861;
   1:  PR[91,2] = PR[90,2] + 7.233;
   1:L PR[91] R[100]mm/sec CNT100;
   1:  PR[91,1] = PR[90,1] + -40.925;
   1:  PR[91,2] = PR[90,2] + 7.096;
   1:L PR[91] R[100]mm/sec CNT100;
   1:  PR[91,1] = PR[90,1] + -42.192;
   1:  PR[91,2] = PR[90,2] + 3.462;
   1:L PR[91] R[100]mm/sec CNT100;
   1:  PR[91,1] = PR[90,1] + -42.239;
   1:  PR[91,2] = PR[90,2] + 3.286;
   1:L PR[91] R[100]mm/sec CNT100;
   1:  PR[91,1] = PR[90,1] + -42.684;
   1:  PR[91,2] = PR[90,2] + -0.752;
   1:L PR[91] R[100]mm/sec CNT100;
   1:  PR[91,1] = PR[90,1] + -42.666;
   1:  PR[91,2] = PR[90,2] + -0.953;
   1:L PR[91] R[100]mm/sec CNT100;
   1:  PR[91,1] = PR[90,1] + -42.240;
   1:  PR[91,2] = PR[90,2] + -4.742;
   1:L PR[91] R[100]mm/sec CNT100;
   1:  PR[91,1] = PR[90,1] + -42.192;
   1:  PR[91,2] = PR[90,2] + -4.921;
   1:L PR[91] R[100]mm/sec CNT100;
   1:  PR[91,1] = PR[90,1] + -40.925;
   1:  PR[91,2] = PR[90,2] + -8.554;
   1:L PR[91] R[100]mm/sec CNT100;
   1:  PR[91,1] = PR[90,1] + -40.861;
   1:  PR[91,2] = PR[90,2] + -8.692;
   1:L PR[91] R[100]mm/sec CNT100;
   1:  PR[91,1] = PR[90,1] + -38.780;
   1:  PR[91,2] = PR[90,2] + -12.014;
   1:L PR[91] R[100]mm/sec CNT100;
   1:  PR[91,1] = PR[90,1] + -38.724;
   1:  PR[91,2] = PR[90,2] + -12.094;
   1:L PR[91] R[100]mm/sec CNT100;
   1:  PR[91,1] = PR[90,1] + -35.829;
   1:  PR[91,2] = PR[90,2] + -15.000;
   1:L PR[91] R[100]mm/sec CNT100;
   1:  PR[91,1] = PR[90,1] + -35.811;
   1:  PR[91,2] = PR[90,2] + -15.013;
   1:L PR[91] R[100]mm/sec CNT100;
   1:  PR[91,1] = PR[90,1] + -32.385;
   1:  PR[91,2] = PR[90,2] + -17.178;
   1:L PR[91] R[100]mm/sec CNT100;
   1:  PR[91,1] = PR[90,1] + -28.515;
   1:  PR[91,2] = PR[90,2] + -18.539;
   1:L PR[91] R[100]mm/sec CNT100;
   1:  PR[91,1] = PR[90,1] + -24.426;
   1:  PR[91,2] = PR[90,2] + -19.024;
   1:L PR[91] R[100]mm/sec CNT100;
   1:  PR[91,1] = PR[90,1] + -20.298;
   1:  PR[91,2] = PR[90,2] + -18.598;
   1:L PR[91] R[100]mm/sec CNT100;
   1:  PR[91,1] = PR[90,1] + -16.362;
   1:  PR[91,2] = PR[90,2] + -17.274;
   1:L PR[91] R[100]mm/sec CNT100;
   1:  PR[91,1] = PR[90,1] + -12.818;
   1:  PR[91,2] = PR[90,2] + -15.111;
   1:L PR[91] R[100]mm/sec CNT100;
   1:  PR[91,1] = PR[90,1] + -9.848;
   1:  PR[91,2] = PR[90,2] + -12.216;
   1:L PR[91] R[100]mm/sec CNT100;
   1:  PR[91,1] = PR[90,1] + -7.605;
   1:  PR[91,2] = PR[90,2] + -8.732;
   1:L PR[91] R[100]mm/sec CNT100;
   1:  PR[91,1] = PR[90,1] + -6.213;
   1:  PR[91,2] = PR[90,2] + -4.840;
   1:L PR[91] R[100]mm/sec CNT100;
   1:  PR[91,1] = PR[90,1] + -5.750;
   1:  PR[91,2] = PR[90,2] + -0.732;
   1:L PR[91] R[100]mm/sec CNT100;
   1:  PR[91,1] = PR[90,1] + -6.135;
   1:  PR[91,2] = PR[90,2] + 2.613;
   1:L PR[91] R[100]mm/sec CNT100TB   .50sec,CALL END_PUD;
   1:  PR[92] = PR[91];
   1:  PR[92,3] = PR[92,3] + 20;
   1:J PR[92] 10% FINE;
   1:  PR[91,1] = PR[90,1] + -88.939;
   1:  PR[91,2] = PR[90,2] + -11.398;
   1:  PR[92] = PR[91];
   1:  PR[92,3] = PR[92,3] + 20;
   1:J PR[92] 10% FINE;
   1:L PR[91] R[100]mm/sec CNT100;
   1:  CALL LASER_DRAHT_START;
   1:  PR[91,1] = PR[90,1] + -86.368;
   1:  PR[91,2] = PR[90,2] + -14.236;
   1:L PR[91] R[100]mm/sec CNT100;
   1:  PR[91,1] = PR[90,1] + -83.249;
   1:  PR[91,2] = PR[90,2] + -16.494;
   1:L PR[91] R[100]mm/sec CNT100;
   1:  PR[91,1] = PR[90,1] + -79.717;
   1:  PR[91,2] = PR[90,2] + -18.073;
   1:L PR[91] R[100]mm/sec CNT100;
   1:  PR[91,1] = PR[90,1] + -75.920;
   1:  PR[91,2] = PR[90,2] + -18.902;
   1:L PR[91] R[100]mm/sec CNT100;
   1:  PR[91,1] = PR[90,1] + -72.026;
   1:  PR[91,2] = PR[90,2] + -18.940;
   1:L PR[91] R[100]mm/sec CNT100;
   1:  PR[91,1] = PR[90,1] + -69.427;
   1:  PR[91,2] = PR[90,2] + -18.416;
   1:L PR[91] R[100]mm/sec CNT100;
   1:  PR[91,1] = PR[90,1] + -68.190;
   1:  PR[91,2] = PR[90,2] + -18.181;
   1:L PR[91] R[100]mm/sec CNT100;
   1:  PR[91,1] = PR[90,1] + -66.042;
   1:  PR[91,2] = PR[90,2] + -17.258;
   1:L PR[91] R[100]mm/sec CNT100;
   1:  PR[91,1] = PR[90,1] + -64.599;
   1:  PR[91,2] = PR[90,2] + -16.655;
   1:L PR[91] R[100]mm/sec CNT100;
   1:  PR[91,1] = PR[90,1] + -62.945;
   1:  PR[91,2] = PR[90,2] + -15.490;
   1:L PR[91] R[100]mm/sec CNT100;
   1:  PR[91,1] = PR[90,1] + -61.397;
   1:  PR[91,2] = PR[90,2] + -14.422;
   1:L PR[91] R[100]mm/sec CNT100;
   1:  PR[91,1] = PR[90,1] + -58.744;
   1:  PR[91,2] = PR[90,2] + -11.582;
   1:L PR[91] R[100]mm/sec CNT100;
   1:  PR[91,1] = PR[90,1] + -56.749;
   1:  PR[91,2] = PR[90,2] + -8.250;
   1:L PR[91] R[100]mm/sec CNT100;
   1:  PR[91,1] = PR[90,1] + -55.514;
   1:  PR[91,2] = PR[90,2] + -4.578;
   1:L PR[91] R[100]mm/sec CNT100;
   1:  PR[91,1] = PR[90,1] + -55.407;
   1:  PR[91,2] = PR[90,2] + -3.591;
   1:L PR[91] R[100]mm/sec CNT100;
   1:  PR[91,1] = PR[90,1] + -55.376;
   1:  PR[91,2] = PR[90,2] + -2.510;
   1:L PR[91] R[100]mm/sec CNT100;
   1:  PR[91,1] = PR[90,1] + -55.203;
   1:  PR[91,2] = PR[90,2] + -0.668;
   1:L PR[91] R[100]mm/sec CNT100;
   1:  PR[91,1] = PR[90,1] + -55.210;
   1:  PR[91,2] = PR[90,2] + -0.437;
   1:L PR[91] R[100]mm/sec CNT100;
   1:  PR[91,1] = PR[90,1] + -55.594;
   1:  PR[91,2] = PR[90,2] + 3.117;
   1:L PR[91] R[100]mm/sec CNT100;
   1:  PR[91,1] = PR[90,1] + -56.822;
   1:  PR[91,2] = PR[90,2] + 6.787;
   1:L PR[91] R[100]mm/sec CNT100;
   1:  PR[91,1] = PR[90,1] + -58.808;
   1:  PR[91,2] = PR[90,2] + 10.117;
   1:L PR[91] R[100]mm/sec CNT100;
   1:  PR[91,1] = PR[90,1] + -61.455;
   1:  PR[91,2] = PR[90,2] + 12.964;
   1:L PR[91] R[100]mm/sec CNT100;
   1:  PR[91,1] = PR[90,1] + -62.398;
   1:  PR[91,2] = PR[90,2] + 13.632;
   1:L PR[91] R[100]mm/sec CNT100;
   1:  PR[91,1] = PR[90,1] + -64.634;
   1:  PR[91,2] = PR[90,2] + 15.192;
   1:L PR[91] R[100]mm/sec CNT100;
   1:  PR[91,1] = PR[90,1] + -68.215;
   1:  PR[91,2] = PR[90,2] + 16.721;
   1:L PR[91] R[100]mm/sec CNT100;
   1:  PR[91,1] = PR[90,1] + -72.030;
   1:  PR[91,2] = PR[90,2] + 17.481;
   1:L PR[91] R[100]mm/sec CNT100;
   1:  PR[91,1] = PR[90,1] + -75.914;
   1:  PR[91,2] = PR[90,2] + 17.445;
   1:L PR[91] R[100]mm/sec CNT100;
   1:  PR[91,1] = PR[90,1] + -79.698;
   1:  PR[91,2] = PR[90,2] + 16.619;
   1:L PR[91] R[100]mm/sec CNT100;
   1:  PR[91,1] = PR[90,1] + -83.220;
   1:  PR[91,2] = PR[90,2] + 15.041;
   1:L PR[91] R[100]mm/sec CNT100;
   1:  PR[91,1] = PR[90,1] + -86.331;
   1:  PR[91,2] = PR[90,2] + 12.784;
   1:L PR[91] R[100]mm/sec CNT100;
   1:  PR[91,1] = PR[90,1] + -88.896;
   1:  PR[91,2] = PR[90,2] + 9.946;
   1:L PR[91] R[100]mm/sec CNT100;
   1:  PR[91,1] = PR[90,1] + -90.810;
   1:  PR[91,2] = PR[90,2] + 6.652;
   1:L PR[91] R[100]mm/sec CNT100;
   1:  PR[91,1] = PR[90,1] + -91.990;
   1:  PR[91,2] = PR[90,2] + 3.041;
   1:L PR[91] R[100]mm/sec CNT100;
   1:  PR[91,1] = PR[90,1] + -92.373;
   1:  PR[91,2] = PR[90,2] + -0.547;
   1:L PR[91] R[100]mm/sec CNT100;
   1:  PR[91,1] = PR[90,1] + -92.432;
   1:  PR[91,2] = PR[90,2] + -0.831;
   1:L PR[91] R[100]mm/sec CNT100;
   1:  PR[91,1] = PR[90,1] + -92.039;
   1:  PR[91,2] = PR[90,2] + -4.496;
   1:L PR[91] R[100]mm/sec CNT100;
   1:  PR[91,1] = PR[90,1] + -90.857;
   1:  PR[91,2] = PR[90,2] + -8.105;
   1:L PR[91] R[100]mm/sec CNT100;
   1:  PR[91,1] = PR[90,1] + -88.939;
   1:  PR[91,2] = PR[90,2] + -11.398;
   1:L PR[91] R[100]mm/sec CNT100TB   .50sec,CALL END_PUD;
   1:  PR[92] = PR[91];
   1:  PR[92,3] = PR[92,3] + 20;
   1:J PR[92] 10% FINE;
   1:  PR[91] = PR[90];
   1:  PR[91,1] = PR[90,1] + 75.472;
   1:  PR[91,2] = PR[90,2] + -19.127;
   1:  PR[91,3] = PR[90,3] + 22.295;
   1:  PR[92] = PR[91];
   1:  PR[92,3] = PR[92,3] + 20;
   1:J PR[92] 10% FINE;
   1:L PR[91] R[100]mm/sec CNT100;
   1:  CALL LASER_DRAHT_START;
   1:  PR[91,1] = PR[90,1] + 77.707;
   1:  PR[91,2] = PR[90,2] + -18.824;
   1:L PR[91] R[100]mm/sec CNT100;
   1:  PR[91,1] = PR[90,1] + 79.977;
   1:  PR[91,2] = PR[90,2] + -18.016;
   1:L PR[91] R[100]mm/sec CNT100;
   1:  PR[91,1] = PR[90,1] + 81.671;
   1:  PR[91,2] = PR[90,2] + -17.392;
   1:L PR[91] R[100]mm/sec CNT100;
   1:  PR[91,1] = PR[90,1] + 83.993;
   1:  PR[91,2] = PR[90,2] + -15.925;
   1:L PR[91] R[100]mm/sec CNT100;
   1:  PR[91,1] = PR[90,1] + 85.202;
   1:  PR[91,2] = PR[90,2] + -15.146;
   1:L PR[91] R[100]mm/sec CNT100;
   1:  PR[91,1] = PR[90,1] + 88.142;
   1:  PR[91,2] = PR[90,2] + -12.194;
   1:L PR[91] R[100]mm/sec CNT100;
   1:  PR[91,1] = PR[90,1] + 90.342;
   1:  PR[91,2] = PR[90,2] + -8.694;
   1:L PR[91] R[100]mm/sec CNT100;
   1:  PR[91,1] = PR[90,1] + 91.704;
   1:  PR[91,2] = PR[90,2] + -4.807;
   1:L PR[91] R[100]mm/sec CNT100;
   1:  PR[91,1] = PR[90,1] + 92.097;
   1:  PR[91,2] = PR[90,2] + -1.400;
   1:L PR[91] R[100]mm/sec CNT100;
   1:  PR[91,1] = PR[90,1] + 92.205;
   1:  PR[91,2] = PR[90,2] + -0.692;
   1:L PR[91] R[100]mm/sec CNT100;
   1:  PR[91,1] = PR[90,1] + 91.906;
   1:  PR[91,2] = PR[90,2] + 1.920;
   1:L PR[91] R[100]mm/sec CNT100;
   1:  PR[91,1] = PR[90,1] + 91.796;
   1:  PR[91,2] = PR[90,2] + 2.516;
   1:L PR[91] R[100]mm/sec CNT100;
   1:  PR[91,1] = PR[90,1] + 91.703;
   1:  PR[91,2] = PR[90,2] + 3.353;
   1:L PR[91] R[100]mm/sec CNT100;
   1:  PR[91,1] = PR[90,1] + 90.342;
   1:  PR[91,2] = PR[90,2] + 7.235;
   1:L PR[91] R[100]mm/sec CNT100;
   1:  PR[91,1] = PR[90,1] + 88.142;
   1:  PR[91,2] = PR[90,2] + 10.735;
   1:L PR[91] R[100]mm/sec CNT100;
   1:  PR[91,1] = PR[90,1] + 85.209;
   1:  PR[91,2] = PR[90,2] + 13.680;
   1:L PR[91] R[100]mm/sec CNT100;
   1:  PR[91,1] = PR[90,1] + 82.872;
   1:  PR[91,2] = PR[90,2] + 15.154;
   1:L PR[91] R[100]mm/sec CNT100;
   1:  PR[91,1] = PR[90,1] + 81.671;
   1:  PR[91,2] = PR[90,2] + 15.930;
   1:L PR[91] R[100]mm/sec CNT100;
   1:  PR[91,1] = PR[90,1] + 79.341;
   1:  PR[91,2] = PR[90,2] + 16.758;
   1:L PR[91] R[100]mm/sec CNT100;
   1:  PR[91,1] = PR[90,1] + 77.707;
   1:  PR[91,2] = PR[90,2] + 17.362;
   1:L PR[91] R[100]mm/sec CNT100;
   1:  PR[91,1] = PR[90,1] + 75.594;
   1:  PR[91,2] = PR[90,2] + 17.620;
   1:L PR[91] R[100]mm/sec CNT100;
   1:  PR[91,1] = PR[90,1] + 73.504;
   1:  PR[91,2] = PR[90,2] + 17.907;
   1:L PR[91] R[100]mm/sec CNT100;
   1:  PR[91,1] = PR[90,1] + 71.787;
   1:  PR[91,2] = PR[90,2] + 17.735;
   1:L PR[91] R[100]mm/sec CNT100;
   1:  PR[91,1] = PR[90,1] + 69.263;
   1:  PR[91,2] = PR[90,2] + 17.523;
   1:L PR[91] R[100]mm/sec CNT100;
   1:  PR[91,1] = PR[90,1] + 68.056;
   1:  PR[91,2] = PR[90,2] + 17.123;
   1:L PR[91] R[100]mm/sec CNT100;
   1:  PR[91,1] = PR[90,1] + 65.192;
   1:  PR[91,2] = PR[90,2] + 16.224;
   1:L PR[91] R[100]mm/sec CNT100;
   1:  PR[91,1] = PR[90,1] + 64.524;
   1:  PR[91,2] = PR[90,2] + 15.821;
   1:L PR[91] R[100]mm/sec CNT100;
   1:  PR[91,1] = PR[90,1] + 61.487;
   1:  PR[91,2] = PR[90,2] + 14.050;
   1:L PR[91] R[100]mm/sec CNT100;
   1:  PR[91,1] = PR[90,1] + 58.354;
   1:  PR[91,2] = PR[90,2] + 11.097;
   1:L PR[91] R[100]mm/sec CNT100;
   1:  PR[91,1] = PR[90,1] + 55.873;
   1:  PR[91,2] = PR[90,2] + 7.525;
   1:L PR[91] R[100]mm/sec CNT100;
   1:  PR[91,1] = PR[90,1] + 54.321;
   1:  PR[91,2] = PR[90,2] + 3.514;
   1:L PR[91] R[100]mm/sec CNT100;
   1:  PR[91,1] = PR[90,1] + 53.882;
   1:  PR[91,2] = PR[90,2] + 0.062;
   1:L PR[91] R[100]mm/sec CNT100;
   1:  PR[91,1] = PR[90,1] + 53.837;
   1:  PR[91,2] = PR[90,2] + -0.667;
   1:L PR[91] R[100]mm/sec CNT100;
   1:  PR[91,1] = PR[90,1] + 54.190;
   1:  PR[91,2] = PR[90,2] + -3.510;
   1:L PR[91] R[100]mm/sec CNT100;
   1:  PR[91,1] = PR[90,1] + 54.254;
   1:  PR[91,2] = PR[90,2] + -4.426;
   1:L PR[91] R[100]mm/sec CNT100;
   1:  PR[91,1] = PR[90,1] + 54.322;
   1:  PR[91,2] = PR[90,2] + -4.976;
   1:L PR[91] R[100]mm/sec CNT100;
   1:  PR[91,1] = PR[90,1] + 55.872;
   1:  PR[91,2] = PR[90,2] + -8.982;
   1:L PR[91] R[100]mm/sec CNT100;
   1:  PR[91,1] = PR[90,1] + 58.317;
   1:  PR[91,2] = PR[90,2] + -12.492;
   1:L PR[91] R[100]mm/sec CNT100;
   1:  PR[91,1] = PR[90,1] + 58.369;
   1:  PR[91,2] = PR[90,2] + -12.571;
   1:L PR[91] R[100]mm/sec CNT100;
   1:  PR[91,1] = PR[90,1] + 61.489;
   1:  PR[91,2] = PR[90,2] + -15.511;
   1:L PR[91] R[100]mm/sec CNT100;
   1:  PR[91,1] = PR[90,1] + 65.193;
   1:  PR[91,2] = PR[90,2] + -17.687;
   1:L PR[91] R[100]mm/sec CNT100;
   1:  PR[91,1] = PR[90,1] + 66.066;
   1:  PR[91,2] = PR[90,2] + -17.975;
   1:L PR[91] R[100]mm/sec CNT100;
   1:  PR[91,1] = PR[90,1] + 69.262;
   1:  PR[91,2] = PR[90,2] + -18.985;
   1:L PR[91] R[100]mm/sec CNT100;
   1:  PR[91,1] = PR[90,1] + 70.738;
   1:  PR[91,2] = PR[90,2] + -19.131;
   1:L PR[91] R[100]mm/sec CNT100;
   1:  PR[91,1] = PR[90,1] + 73.504;
   1:  PR[91,2] = PR[90,2] + -19.369;
   1:L PR[91] R[100]mm/sec CNT100;
   1:  PR[91,1] = PR[90,1] + 75.472;
   1:  PR[91,2] = PR[90,2] + -19.127;
   1:L PR[91] R[100]mm/sec CNT100TB   .50sec,CALL END_PUD;
   1:  PR[92] = PR[91];
   1:  PR[92,3] = PR[92,3] + 20;
   1:J PR[92] 10% FINE;
   1:  PR[91,1] = PR[90,1] + 37.828;
   1:  PR[91,2] = PR[90,2] + -13.861;
   1:  PR[92] = PR[91];
   1:  PR[92,3] = PR[92,3] + 20;
   1:J PR[92] 10% FINE;
   1:L PR[91] R[100]mm/sec CNT100;
   1:  CALL LASER_DRAHT_START;
   1:  PR[91,1] = PR[90,1] + 37.858;
   1:  PR[91,2] = PR[90,2] + -13.831;
   1:L PR[91] R[100]mm/sec CNT100;
   1:  PR[91,1] = PR[90,1] + 40.722;
   1:  PR[91,2] = PR[90,2] + -10.089;
   1:L PR[91] R[100]mm/sec CNT100;
   1:  PR[91,1] = PR[90,1] + 40.785;
   1:  PR[91,2] = PR[90,2] + -9.999;
   1:L PR[91] R[100]mm/sec CNT100;
   1:  PR[91,1] = PR[90,1] + 40.830;
   1:  PR[91,2] = PR[90,2] + -9.903;
   1:L PR[91] R[100]mm/sec CNT100;
   1:  PR[91,1] = PR[90,1] + 42.623;
   1:  PR[91,2] = PR[90,2] + -5.565;
   1:L PR[91] R[100]mm/sec CNT100;
   1:  PR[91,1] = PR[90,1] + 42.638;
   1:  PR[91,2] = PR[90,2] + -5.509;
   1:L PR[91] R[100]mm/sec CNT100;
   1:  PR[91,1] = PR[90,1] + 42.845;
   1:  PR[91,2] = PR[90,2] + -3.661;
   1:L PR[91] R[100]mm/sec CNT100;
   1:  PR[91,1] = PR[90,1] + 43.245;
   1:  PR[91,2] = PR[90,2] + -0.613;
   1:L PR[91] R[100]mm/sec CNT100;
   1:  PR[91,1] = PR[90,1] + 43.244;
   1:  PR[91,2] = PR[90,2] + -0.541;
   1:L PR[91] R[100]mm/sec CNT100;
   1:  PR[91,1] = PR[90,1] + 42.643;
   1:  PR[91,2] = PR[90,2] + 4.031;
   1:L PR[91] R[100]mm/sec CNT100;
   1:  PR[91,1] = PR[90,1] + 42.623;
   1:  PR[91,2] = PR[90,2] + 4.106;
   1:L PR[91] R[100]mm/sec CNT100;
   1:  PR[91,1] = PR[90,1] + 40.830;
   1:  PR[91,2] = PR[90,2] + 8.444;
   1:L PR[91] R[100]mm/sec CNT100;
   1:  PR[91,1] = PR[90,1] + 40.785;
   1:  PR[91,2] = PR[90,2] + 8.540;
   1:L PR[91] R[100]mm/sec CNT100;
   1:  PR[91,1] = PR[90,1] + 40.722;
   1:  PR[91,2] = PR[90,2] + 8.630;
   1:L PR[91] R[100]mm/sec CNT100;
   1:  PR[91,1] = PR[90,1] + 37.858;
   1:  PR[91,2] = PR[90,2] + 12.372;
   1:L PR[91] R[100]mm/sec CNT100;
   1:  PR[91,1] = PR[90,1] + 37.828;
   1:  PR[91,2] = PR[90,2] + 12.402;
   1:L PR[91] R[100]mm/sec CNT100;
   1:  PR[91,1] = PR[90,1] + 34.053;
   1:  PR[91,2] = PR[90,2] + 15.305;
   1:L PR[91] R[100]mm/sec CNT100;
   1:  PR[91,1] = PR[90,1] + 34.005;
   1:  PR[91,2] = PR[90,2] + 15.339;
   1:L PR[91] R[100]mm/sec CNT100;
   1:  PR[91,1] = PR[90,1] + 33.950;
   1:  PR[91,2] = PR[90,2] + 15.364;
   1:L PR[91] R[100]mm/sec CNT100;
   1:  PR[91,1] = PR[90,1] + 29.532;
   1:  PR[91,2] = PR[90,2] + 17.202;
   1:L PR[91] R[100]mm/sec CNT100;
   1:  PR[91,1] = PR[90,1] + 24.725;
   1:  PR[91,2] = PR[90,2] + 17.835;
   1:L PR[91] R[100]mm/sec CNT100;
   1:  PR[91,1] = PR[90,1] + 19.917;
   1:  PR[91,2] = PR[90,2] + 17.218;
   1:L PR[91] R[100]mm/sec CNT100;
   1:  PR[91,1] = PR[90,1] + 15.434;
   1:  PR[91,2] = PR[90,2] + 15.363;
   1:L PR[91] R[100]mm/sec CNT100;
   1:  PR[91,1] = PR[90,1] + 11.576;
   1:  PR[91,2] = PR[90,2] + 12.419;
   1:L PR[91] R[100]mm/sec CNT100;
   1:  PR[91,1] = PR[90,1] + 8.618;
   1:  PR[91,2] = PR[90,2] + 8.572;
   1:L PR[91] R[100]mm/sec CNT100;
   1:  PR[91,1] = PR[90,1] + 6.753;
   1:  PR[91,2] = PR[90,2] + 4.054;
   1:L PR[91] R[100]mm/sec CNT100;
   1:  PR[91,1] = PR[90,1] + 6.129;
   1:  PR[91,2] = PR[90,2] + -0.790;
   1:L PR[91] R[100]mm/sec CNT100;
   1:  PR[91,1] = PR[90,1] + 6.770;
   1:  PR[91,2] = PR[90,2] + -5.576;
   1:L PR[91] R[100]mm/sec CNT100;
   1:  PR[91,1] = PR[90,1] + 8.618;
   1:  PR[91,2] = PR[90,2] + -10.029;
   1:L PR[91] R[100]mm/sec CNT100;
   1:  PR[91,1] = PR[90,1] + 11.576;
   1:  PR[91,2] = PR[90,2] + -13.878;
   1:L PR[91] R[100]mm/sec CNT100;
   1:  PR[91,1] = PR[90,1] + 15.434;
   1:  PR[91,2] = PR[90,2] + -16.822;
   1:L PR[91] R[100]mm/sec CNT100;
   1:  PR[91,1] = PR[90,1] + 19.917;
   1:  PR[91,2] = PR[90,2] + -18.677;
   1:L PR[91] R[100]mm/sec CNT100;
   1:  PR[91,1] = PR[90,1] + 24.725;
   1:  PR[91,2] = PR[90,2] + -19.294;
   1:L PR[91] R[100]mm/sec CNT100;
   1:  PR[91,1] = PR[90,1] + 29.531;
   1:  PR[91,2] = PR[90,2] + -18.661;
   1:L PR[91] R[100]mm/sec CNT100;
   1:  PR[91,1] = PR[90,1] + 34.038;
   1:  PR[91,2] = PR[90,2] + -16.774;
   1:L PR[91] R[100]mm/sec CNT100;
   1:  PR[91,1] = PR[90,1] + 34.053;
   1:  PR[91,2] = PR[90,2] + -16.764;
   1:L PR[91] R[100]mm/sec CNT100;
   1:  PR[91,1] = PR[90,1] + 37.828;
   1:  PR[91,2] = PR[90,2] + -13.861;
   1:L PR[91] R[100]mm/sec CNT100TB   .50sec,CALL END_PUD;
   1:  PR[92] = PR[91];
   1:  PR[92,3] = PR[92,3] + 20;
   1:J PR[92] 10% FINE;
   1:  PR[91,1] = PR[90,1] + -5.907;
   1:  PR[91,2] = PR[90,2] + 3.403;
   1:  PR[92] = PR[91];
   1:  PR[92,3] = PR[92,3] + 20;
   1:J PR[92] 10% FINE;
   1:L PR[91] R[100]mm/sec CNT100;
   1:  CALL LASER_DRAHT_START;
   1:  PR[91,1] = PR[90,1] + -7.311;
   1:  PR[91,2] = PR[90,2] + 7.321;
   1:L PR[91] R[100]mm/sec CNT100;
   1:  PR[91,1] = PR[90,1] + -9.571;
   1:  PR[91,2] = PR[90,2] + 10.825;
   1:L PR[91] R[100]mm/sec CNT100;
   1:  PR[91,1] = PR[90,1] + -11.755;
   1:  PR[91,2] = PR[90,2] + 12.959;
   1:L PR[91] R[100]mm/sec CNT100;
   1:  PR[91,1] = PR[90,1] + -12.555;
   1:  PR[91,2] = PR[90,2] + 13.729;
   1:L PR[91] R[100]mm/sec CNT100;
   1:  PR[91,1] = PR[90,1] + -16.126;
   1:  PR[91,2] = PR[90,2] + 15.902;
   1:L PR[91] R[100]mm/sec CNT100;
   1:  PR[91,1] = PR[90,1] + -20.084;
   1:  PR[91,2] = PR[90,2] + 17.228;
   1:L PR[91] R[100]mm/sec CNT100;
   1:  PR[91,1] = PR[90,1] + -24.232;
   1:  PR[91,2] = PR[90,2] + 17.652;
   1:L PR[91] R[100]mm/sec CNT100;
   1:  PR[91,1] = PR[90,1] + -28.362;
   1:  PR[91,2] = PR[90,2] + 17.152;
   1:L PR[91] R[100]mm/sec CNT100;
   1:  PR[91,1] = PR[90,1] + -32.270;
   1:  PR[91,2] = PR[90,2] + 15.765;
   1:L PR[91] R[100]mm/sec CNT100;
   1:  PR[91,1] = PR[90,1] + -35.763;
   1:  PR[91,2] = PR[90,2] + 13.559;
   1:L PR[91] R[100]mm/sec CNT100;
   1:  PR[91,1] = PR[90,1] + -38.670;
   1:  PR[91,2] = PR[90,2] + 10.652;
   1:L PR[91] R[100]mm/sec CNT100;
   1:  PR[91,1] = PR[90,1] + -40.850;
   1:  PR[91,2] = PR[90,2] + 7.164;
   1:L PR[91] R[100]mm/sec CNT100;
   1:  PR[91,1] = PR[90,1] + -42.189;
   1:  PR[91,2] = PR[90,2] + 3.308;
   1:L PR[91] R[100]mm/sec CNT100;
   1:  PR[91,1] = PR[90,1] + -42.641;
   1:  PR[91,2] = PR[90,2] + -0.729;
   1:L PR[91] R[100]mm/sec CNT100;
   1:  PR[91,1] = PR[90,1] + -42.189;
   1:  PR[91,2] = PR[90,2] + -4.766;
   1:L PR[91] R[100]mm/sec CNT100;
   1:  PR[91,1] = PR[90,1] + -40.831;
   1:  PR[91,2] = PR[90,2] + -8.665;
   1:L PR[91] R[100]mm/sec CNT100;
   1:  PR[91,1] = PR[90,1] + -38.998;
   1:  PR[91,2] = PR[90,2] + -11.590;
   1:L PR[91] R[100]mm/sec CNT100;
   1:  PR[91,1] = PR[90,1] + -38.672;
   1:  PR[91,2] = PR[90,2] + -12.108;
   1:L PR[91] R[100]mm/sec CNT100;
   1:  PR[91,1] = PR[90,1] + -35.763;
   1:  PR[91,2] = PR[90,2] + -15.018;
   1:L PR[91] R[100]mm/sec CNT100;
   1:  PR[91,1] = PR[90,1] + -32.270;
   1:  PR[91,2] = PR[90,2] + -17.224;
   1:L PR[91] R[100]mm/sec CNT100;
   1:  PR[91,1] = PR[90,1] + -28.362;
   1:  PR[91,2] = PR[90,2] + -18.611;
   1:L PR[91] R[100]mm/sec CNT100;
   1:  PR[91,1] = PR[90,1] + -24.232;
   1:  PR[91,2] = PR[90,2] + -19.110;
   1:L PR[91] R[100]mm/sec CNT100;
   1:  PR[91,1] = PR[90,1] + -20.084;
   1:  PR[91,2] = PR[90,2] + -18.687;
   1:L PR[91] R[100]mm/sec CNT100;
   1:  PR[91,1] = PR[90,1] + -16.126;
   1:  PR[91,2] = PR[90,2] + -17.361;
   1:L PR[91] R[100]mm/sec CNT100;
   1:  PR[91,1] = PR[90,1] + -12.560;
   1:  PR[91,2] = PR[90,2] + -15.190;
   1:L PR[91] R[100]mm/sec CNT100;
   1:  PR[91,1] = PR[90,1] + -9.570;
   1:  PR[91,2] = PR[90,2] + -12.282;
   1:L PR[91] R[100]mm/sec CNT100;
   1:  PR[91,1] = PR[90,1] + -7.311;
   1:  PR[91,2] = PR[90,2] + -8.780;
   1:L PR[91] R[100]mm/sec CNT100;
   1:  PR[91,1] = PR[90,1] + -5.907;
   1:  PR[91,2] = PR[90,2] + -4.862;
   1:L PR[91] R[100]mm/sec CNT100;
   1:  PR[91,1] = PR[90,1] + -5.600;
   1:  PR[91,2] = PR[90,2] + -2.198;
   1:L PR[91] R[100]mm/sec CNT100;
   1:  PR[91,1] = PR[90,1] + -5.449;
   1:  PR[91,2] = PR[90,2] + -0.741;
   1:L PR[91] R[100]mm/sec CNT100;
   1:  PR[91,1] = PR[90,1] + -5.760;
   1:  PR[91,2] = PR[90,2] + 1.963;
   1:L PR[91] R[100]mm/sec CNT100;
   1:  PR[91,1] = PR[90,1] + -5.755;
   1:  PR[91,2] = PR[90,2] + 2.095;
   1:L PR[91] R[100]mm/sec CNT100;
   1:  PR[91,1] = PR[90,1] + -5.907;
   1:  PR[91,2] = PR[90,2] + 3.403;
   1:L PR[91] R[100]mm/sec CNT100TB   .50sec,CALL END_PUD;
   1:  PR[92] = PR[91];
   1:  PR[92,3] = PR[92,3] + 20;
   1:J PR[92] 10% FINE;
   1:  PR[91,1] = PR[90,1] + -73.284;
   1:  PR[91,2] = PR[90,2] + -18.980;
   1:  PR[92] = PR[91];
   1:  PR[92,3] = PR[92,3] + 20;
   1:J PR[92] 10% FINE;
   1:L PR[91] R[100]mm/sec CNT100;
   1:  CALL LASER_DRAHT_START;
   1:  PR[91,1] = PR[90,1] + -71.769;
   1:  PR[91,2] = PR[90,2] + -19.006;
   1:L PR[91] R[100]mm/sec CNT100;
   1:  PR[91,1] = PR[90,1] + -69.726;
   1:  PR[91,2] = PR[90,2] + -18.595;
   1:L PR[91] R[100]mm/sec CNT100;
   1:  PR[91,1] = PR[90,1] + -67.925;
   1:  PR[91,2] = PR[90,2] + -18.251;
   1:L PR[91] R[100]mm/sec CNT100;
   1:  PR[91,1] = PR[90,1] + -66.320;
   1:  PR[91,2] = PR[90,2] + -17.562;
   1:L PR[91] R[100]mm/sec CNT100;
   1:  PR[91,1] = PR[90,1] + -64.309;
   1:  PR[91,2] = PR[90,2] + -16.722;
   1:L PR[91] R[100]mm/sec CNT100;
   1:  PR[91,1] = PR[90,1] + -61.097;
   1:  PR[91,2] = PR[90,2] + -14.488;
   1:L PR[91] R[100]mm/sec CNT100;
   1:  PR[91,1] = PR[90,1] + -58.423;
   1:  PR[91,2] = PR[90,2] + -11.634;
   1:L PR[91] R[100]mm/sec CNT100;
   1:  PR[91,1] = PR[90,1] + -56.415;
   1:  PR[91,2] = PR[90,2] + -8.288;
   1:L PR[91] R[100]mm/sec CNT100;
   1:  PR[91,1] = PR[90,1] + -55.171;
   1:  PR[91,2] = PR[90,2] + -4.598;
   1:L PR[91] R[100]mm/sec CNT100;
   1:  PR[91,1] = PR[90,1] + -55.146;
   1:  PR[91,2] = PR[90,2] + -4.367;
   1:L PR[91] R[100]mm/sec CNT100;
   1:  PR[91,1] = PR[90,1] + -55.133;
   1:  PR[91,2] = PR[90,2] + -3.930;
   1:L PR[91] R[100]mm/sec CNT100;
   1:  PR[91,1] = PR[90,1] + -54.982;
   1:  PR[91,2] = PR[90,2] + -2.318;
   1:L PR[91] R[100]mm/sec CNT100;
   1:  PR[91,1] = PR[90,1] + -54.806;
   1:  PR[91,2] = PR[90,2] + -0.730;
   1:L PR[91] R[100]mm/sec CNT100;
   1:  PR[91,1] = PR[90,1] + -55.066;
   1:  PR[91,2] = PR[90,2] + 1.610;
   1:L PR[91] R[100]mm/sec CNT100;
   1:  PR[91,1] = PR[90,1] + -55.209;
   1:  PR[91,2] = PR[90,2] + 3.143;
   1:L PR[91] R[100]mm/sec CNT100;
   1:  PR[91,1] = PR[90,1] + -56.479;
   1:  PR[91,2] = PR[90,2] + 6.801;
   1:L PR[91] R[100]mm/sec CNT100;
   1:  PR[91,1] = PR[90,1] + -57.361;
   1:  PR[91,2] = PR[90,2] + 8.225;
   1:L PR[91] R[100]mm/sec CNT100;
   1:  PR[91,1] = PR[90,1] + -58.520;
   1:  PR[91,2] = PR[90,2] + 10.165;
   1:L PR[91] R[100]mm/sec CNT100;
   1:  PR[91,1] = PR[90,1] + -61.179;
   1:  PR[91,2] = PR[90,2] + 13.018;
   1:L PR[91] R[100]mm/sec CNT100;
   1:  PR[91,1] = PR[90,1] + -64.384;
   1:  PR[91,2] = PR[90,2] + 15.258;
   1:L PR[91] R[100]mm/sec CNT100;
   1:  PR[91,1] = PR[90,1] + -65.098;
   1:  PR[91,2] = PR[90,2] + 15.567;
   1:L PR[91] R[100]mm/sec CNT100;
   1:  PR[91,1] = PR[90,1] + -67.972;
   1:  PR[91,2] = PR[90,2] + 16.784;
   1:L PR[91] R[100]mm/sec CNT100;
   1:  PR[91,1] = PR[90,1] + -71.804;
   1:  PR[91,2] = PR[90,2] + 17.542;
   1:L PR[91] R[100]mm/sec CNT100;
   1:  PR[91,1] = PR[90,1] + -75.700;
   1:  PR[91,2] = PR[90,2] + 17.502;
   1:L PR[91] R[100]mm/sec CNT100;
   1:  PR[91,1] = PR[90,1] + -79.495;
   1:  PR[91,2] = PR[90,2] + 16.669;
   1:L PR[91] R[100]mm/sec CNT100;
   1:  PR[91,1] = PR[90,1] + -83.026;
   1:  PR[91,2] = PR[90,2] + 15.084;
   1:L PR[91] R[100]mm/sec CNT100;
   1:  PR[91,1] = PR[90,1] + -86.143;
   1:  PR[91,2] = PR[90,2] + 12.819;
   1:L PR[91] R[100]mm/sec CNT100;
   1:  PR[91,1] = PR[90,1] + -88.713;
   1:  PR[91,2] = PR[90,2] + 9.972;
   1:L PR[91] R[100]mm/sec CNT100;
   1:  PR[91,1] = PR[90,1] + -90.630;
   1:  PR[91,2] = PR[90,2] + 6.669;
   1:L PR[91] R[100]mm/sec CNT100;
   1:  PR[91,1] = PR[90,1] + -91.812;
   1:  PR[91,2] = PR[90,2] + 3.050;
   1:L PR[91] R[100]mm/sec CNT100;
   1:  PR[91,1] = PR[90,1] + -92.142;
   1:  PR[91,2] = PR[90,2] + -0.042;
   1:L PR[91] R[100]mm/sec CNT100;
   1:  PR[91,1] = PR[90,1] + -92.239;
   1:  PR[91,2] = PR[90,2] + -0.499;
   1:L PR[91] R[100]mm/sec CNT100;
   1:  PR[91,1] = PR[90,1] + -92.281;
   1:  PR[91,2] = PR[90,2] + -0.775;
   1:L PR[91] R[100]mm/sec CNT100;
   1:  PR[91,1] = PR[90,1] + -91.994;
   1:  PR[91,2] = PR[90,2] + -3.473;
   1:L PR[91] R[100]mm/sec CNT100;
   1:  PR[91,1] = PR[90,1] + -91.876;
   1:  PR[91,2] = PR[90,2] + -4.160;
   1:L PR[91] R[100]mm/sec CNT100;
   1:  PR[91,1] = PR[90,1] + -91.840;
   1:  PR[91,2] = PR[90,2] + -4.508;
   1:L PR[91] R[100]mm/sec CNT100;
   1:  PR[91,1] = PR[90,1] + -90.762;
   1:  PR[91,2] = PR[90,2] + -7.799;
   1:L PR[91] R[100]mm/sec CNT100;
   1:  PR[91,1] = PR[90,1] + -90.655;
   1:  PR[91,2] = PR[90,2] + -8.126;
   1:L PR[91] R[100]mm/sec CNT100;
   1:  PR[91,1] = PR[90,1] + -88.735;
   1:  PR[91,2] = PR[90,2] + -11.427;
   1:L PR[91] R[100]mm/sec CNT100;
   1:  PR[91,1] = PR[90,1] + -86.158;
   1:  PR[91,2] = PR[90,2] + -14.274;
   1:L PR[91] R[100]mm/sec CNT100;
   1:  PR[91,1] = PR[90,1] + -83.032;
   1:  PR[91,2] = PR[90,2] + -16.541;
   1:L PR[91] R[100]mm/sec CNT100;
   1:  PR[91,1] = PR[90,1] + -79.491;
   1:  PR[91,2] = PR[90,2] + -18.128;
   1:L PR[91] R[100]mm/sec CNT100;
   1:  PR[91,1] = PR[90,1] + -75.686;
   1:  PR[91,2] = PR[90,2] + -18.963;
   1:L PR[91] R[100]mm/sec CNT100;
   1:  PR[91,1] = PR[90,1] + -73.284;
   1:  PR[91,2] = PR[90,2] + -18.980;
   1:L PR[91] R[100]mm/sec CNT100TB   .50sec,CALL END_PUD;
   1:  PR[92] = PR[91];
   1:  PR[92,3] = PR[92,3] + 20;
   1:J PR[92] 10% FINE;
   1:  PR[91] = PR[90];
   1:  PR[91,1] = PR[90,1] + 73.272;
   1:  PR[91,2] = PR[90,2] + -19.473;
   1:  PR[91,3] = PR[90,3] + 23.595;
   1:  PR[92] = PR[91];
   1:  PR[92,3] = PR[92,3] + 20;
   1:J PR[92] 10% FINE;
   1:L PR[91] R[100]mm/sec CNT100;
   1:  CALL LASER_DRAHT_START;
   1:  PR[91,1] = PR[90,1] + 74.511;
   1:  PR[91,2] = PR[90,2] + -19.321;
   1:L PR[91] R[100]mm/sec CNT100;
   1:  PR[91,1] = PR[90,1] + 77.495;
   1:  PR[91,2] = PR[90,2] + -18.917;
   1:L PR[91] R[100]mm/sec CNT100;
   1:  PR[91,1] = PR[90,1] + 79.122;
   1:  PR[91,2] = PR[90,2] + -18.338;
   1:L PR[91] R[100]mm/sec CNT100;
   1:  PR[91,1] = PR[90,1] + 81.475;
   1:  PR[91,2] = PR[90,2] + -17.471;
   1:L PR[91] R[100]mm/sec CNT100;
   1:  PR[91,1] = PR[90,1] + 83.259;
   1:  PR[91,2] = PR[90,2] + -16.344;
   1:L PR[91] R[100]mm/sec CNT100;
   1:  PR[91,1] = PR[90,1] + 85.018;
   1:  PR[91,2] = PR[90,2] + -15.210;
   1:L PR[91] R[100]mm/sec CNT100;
   1:  PR[91,1] = PR[90,1] + 87.967;
   1:  PR[91,2] = PR[90,2] + -12.243;
   1:L PR[91] R[100]mm/sec CNT100;
   1:  PR[91,1] = PR[90,1] + 90.174;
   1:  PR[91,2] = PR[90,2] + -8.726;
   1:L PR[91] R[100]mm/sec CNT100;
   1:  PR[91,1] = PR[90,1] + 91.540;
   1:  PR[91,2] = PR[90,2] + -4.823;
   1:L PR[91] R[100]mm/sec CNT100;
   1:  PR[91,1] = PR[90,1] + 91.871;
   1:  PR[91,2] = PR[90,2] + -1.951;
   1:L PR[91] R[100]mm/sec CNT100;
   1:  PR[91,1] = PR[90,1] + 92.063;
   1:  PR[91,2] = PR[90,2] + -0.692;
   1:L PR[91] R[100]mm/sec CNT100;
   1:  PR[91,1] = PR[90,1] + 91.859;
   1:  PR[91,2] = PR[90,2] + 1.092;
   1:L PR[91] R[100]mm/sec CNT100;
   1:  PR[91,1] = PR[90,1] + 91.690;
   1:  PR[91,2] = PR[90,2] + 2.004;
   1:L PR[91] R[100]mm/sec CNT100;
   1:  PR[91,1] = PR[90,1] + 91.538;
   1:  PR[91,2] = PR[90,2] + 3.369;
   1:L PR[91] R[100]mm/sec CNT100;
   1:  PR[91,1] = PR[90,1] + 90.174;
   1:  PR[91,2] = PR[90,2] + 7.267;
   1:L PR[91] R[100]mm/sec CNT100;
   1:  PR[91,1] = PR[90,1] + 87.967;
   1:  PR[91,2] = PR[90,2] + 10.784;
   1:L PR[91] R[100]mm/sec CNT100;
   1:  PR[91,1] = PR[90,1] + 85.025;
   1:  PR[91,2] = PR[90,2] + 13.744;
   1:L PR[91] R[100]mm/sec CNT100;
   1:  PR[91,1] = PR[90,1] + 83.157;
   1:  PR[91,2] = PR[90,2] + 14.922;
   1:L PR[91] R[100]mm/sec CNT100;
   1:  PR[91,1] = PR[90,1] + 81.475;
   1:  PR[91,2] = PR[90,2] + 16.009;
   1:L PR[91] R[100]mm/sec CNT100;
   1:  PR[91,1] = PR[90,1] + 79.690;
   1:  PR[91,2] = PR[90,2] + 16.643;
   1:L PR[91] R[100]mm/sec CNT100;
   1:  PR[91,1] = PR[90,1] + 77.495;
   1:  PR[91,2] = PR[90,2] + 17.456;
   1:L PR[91] R[100]mm/sec CNT100;
   1:  PR[91,1] = PR[90,1] + 75.986;
   1:  PR[91,2] = PR[90,2] + 17.640;
   1:L PR[91] R[100]mm/sec CNT100;
   1:  PR[91,1] = PR[90,1] + 73.270;
   1:  PR[91,2] = PR[90,2] + 18.012;
   1:L PR[91] R[100]mm/sec CNT100;
   1:  PR[91,1] = PR[90,1] + 72.197;
   1:  PR[91,2] = PR[90,2] + 17.905;
   1:L PR[91] R[100]mm/sec CNT100;
   1:  PR[91,1] = PR[90,1] + 69.002;
   1:  PR[91,2] = PR[90,2] + 17.636;
   1:L PR[91] R[100]mm/sec CNT100;
   1:  PR[91,1] = PR[90,1] + 68.451;
   1:  PR[91,2] = PR[90,2] + 17.453;
   1:L PR[91] R[100]mm/sec CNT100;
   1:  PR[91,1] = PR[90,1] + 64.888;
   1:  PR[91,2] = PR[90,2] + 16.335;
   1:L PR[91] R[100]mm/sec CNT100;
   1:  PR[91,1] = PR[90,1] + 63.034;
   1:  PR[91,2] = PR[90,2] + 15.250;
   1:L PR[91] R[100]mm/sec CNT100;
   1:  PR[91,1] = PR[90,1] + 61.049;
   1:  PR[91,2] = PR[90,2] + 14.153;
   1:L PR[91] R[100]mm/sec CNT100;
   1:  PR[91,1] = PR[90,1] + 58.225;
   1:  PR[91,2] = PR[90,2] + 11.615;
   1:L PR[91] R[100]mm/sec CNT100;
   1:  PR[91,1] = PR[90,1] + 57.749;
   1:  PR[91,2] = PR[90,2] + 11.204;
   1:L PR[91] R[100]mm/sec CNT100;
   1:  PR[91,1] = PR[90,1] + 55.897;
   1:  PR[91,2] = PR[90,2] + 8.536;
   1:L PR[91] R[100]mm/sec CNT100;
   1:  PR[91,1] = PR[90,1] + 55.238;
   1:  PR[91,2] = PR[90,2] + 7.619;
   1:L PR[91] R[100]mm/sec CNT100;
   1:  PR[91,1] = PR[90,1] + 54.224;
   1:  PR[91,2] = PR[90,2] + 4.984;
   1:L PR[91] R[100]mm/sec CNT100;
   1:  PR[91,1] = PR[90,1] + 53.660;
   1:  PR[91,2] = PR[90,2] + 3.563;
   1:L PR[91] R[100]mm/sec CNT100;
   1:  PR[91,1] = PR[90,1] + 53.352;
   1:  PR[91,2] = PR[90,2] + 1.137;
   1:L PR[91] R[100]mm/sec CNT100;
   1:  PR[91,1] = PR[90,1] + 53.240;
   1:  PR[91,2] = PR[90,2] + -0.667;
   1:L PR[91] R[100]mm/sec CNT100;
   1:  PR[91,1] = PR[90,1] + 53.292;
   1:  PR[91,2] = PR[90,2] + -1.083;
   1:L PR[91] R[100]mm/sec CNT100;
   1:  PR[91,1] = PR[90,1] + 53.446;
   1:  PR[91,2] = PR[90,2] + -3.288;
   1:L PR[91] R[100]mm/sec CNT100;
   1:  PR[91,1] = PR[90,1] + 53.662;
   1:  PR[91,2] = PR[90,2] + -5.031;
   1:L PR[91] R[100]mm/sec CNT100;
   1:  PR[91,1] = PR[90,1] + 55.241;
   1:  PR[91,2] = PR[90,2] + -9.088;
   1:L PR[91] R[100]mm/sec CNT100;
   1:  PR[91,1] = PR[90,1] + 57.194;
   1:  PR[91,2] = PR[90,2] + -11.892;
   1:L PR[91] R[100]mm/sec CNT100;
   1:  PR[91,1] = PR[90,1] + 57.748;
   1:  PR[91,2] = PR[90,2] + -12.667;
   1:L PR[91] R[100]mm/sec CNT100;
   1:  PR[91,1] = PR[90,1] + 61.046;
   1:  PR[91,2] = PR[90,2] + -15.610;
   1:L PR[91] R[100]mm/sec CNT100;
   1:  PR[91,1] = PR[90,1] + 63.034;
   1:  PR[91,2] = PR[90,2] + -16.709;
   1:L PR[91] R[100]mm/sec CNT100;
   1:  PR[91,1] = PR[90,1] + 64.891;
   1:  PR[91,2] = PR[90,2] + -17.795;
   1:L PR[91] R[100]mm/sec CNT100;
   1:  PR[91,1] = PR[90,1] + 68.993;
   1:  PR[91,2] = PR[90,2] + -19.095;
   1:L PR[91] R[100]mm/sec CNT100;
   1:  PR[91,1] = PR[90,1] + 73.272;
   1:  PR[91,2] = PR[90,2] + -19.473;
   1:L PR[91] R[100]mm/sec CNT100TB   .50sec,CALL END_PUD;
   1:  PR[92] = PR[91];
   1:  PR[92,3] = PR[92,3] + 20;
   1:J PR[92] 10% FINE;
   1:  PR[91,1] = PR[90,1] + 34.001;
   1:  PR[91,2] = PR[90,2] + 15.387;
   1:  PR[92] = PR[91];
   1:  PR[92,3] = PR[92,3] + 20;
   1:J PR[92] 10% FINE;
   1:L PR[91] R[100]mm/sec CNT100;
   1:  CALL LASER_DRAHT_START;
   1:  PR[91,1] = PR[90,1] + 29.511;
   1:  PR[91,2] = PR[90,2] + 17.264;
   1:L PR[91] R[100]mm/sec CNT100;
   1:  PR[91,1] = PR[90,1] + 24.682;
   1:  PR[91,2] = PR[90,2] + 17.919;
   1:L PR[91] R[100]mm/sec CNT100;
   1:  PR[91,1] = PR[90,1] + 19.849;
   1:  PR[91,2] = PR[90,2] + 17.301;
   1:L PR[91] R[100]mm/sec CNT100;
   1:  PR[91,1] = PR[90,1] + 15.329;
   1:  PR[91,2] = PR[90,2] + 15.450;
   1:L PR[91] R[100]mm/sec CNT100;
   1:  PR[91,1] = PR[90,1] + 11.444;
   1:  PR[91,2] = PR[90,2] + 12.492;
   1:L PR[91] R[100]mm/sec CNT100;
   1:  PR[91,1] = PR[90,1] + 8.460;
   1:  PR[91,2] = PR[90,2] + 8.624;
   1:L PR[91] R[100]mm/sec CNT100;
   1:  PR[91,1] = PR[90,1] + 6.582;
   1:  PR[91,2] = PR[90,2] + 4.114;
   1:L PR[91] R[100]mm/sec CNT100;
   1:  PR[91,1] = PR[90,1] + 5.940;
   1:  PR[91,2] = PR[90,2] + -0.729;
   1:L PR[91] R[100]mm/sec CNT100;
   1:  PR[91,1] = PR[90,1] + 6.582;
   1:  PR[91,2] = PR[90,2] + -5.573;
   1:L PR[91] R[100]mm/sec CNT100;
   1:  PR[91,1] = PR[90,1] + 8.460;
   1:  PR[91,2] = PR[90,2] + -10.084;
   1:L PR[91] R[100]mm/sec CNT100;
   1:  PR[91,1] = PR[90,1] + 11.445;
   1:  PR[91,2] = PR[90,2] + -13.951;
   1:L PR[91] R[100]mm/sec CNT100;
   1:  PR[91,1] = PR[90,1] + 15.330;
   1:  PR[91,2] = PR[90,2] + -16.909;
   1:L PR[91] R[100]mm/sec CNT100;
   1:  PR[91,1] = PR[90,1] + 19.846;
   1:  PR[91,2] = PR[90,2] + -18.759;
   1:L PR[91] R[100]mm/sec CNT100;
   1:  PR[91,1] = PR[90,1] + 24.683;
   1:  PR[91,2] = PR[90,2] + -19.377;
   1:L PR[91] R[100]mm/sec CNT100;
   1:  PR[91,1] = PR[90,1] + 29.511;
   1:  PR[91,2] = PR[90,2] + -18.723;
   1:L PR[91] R[100]mm/sec CNT100;
   1:  PR[91,1] = PR[90,1] + 34.002;
   1:  PR[91,2] = PR[90,2] + -16.846;
   1:L PR[91] R[100]mm/sec CNT100;
   1:  PR[91,1] = PR[90,1] + 37.853;
   1:  PR[91,2] = PR[90,2] + -13.877;
   1:L PR[91] R[100]mm/sec CNT100;
   1:  PR[91,1] = PR[90,1] + 40.801;
   1:  PR[91,2] = PR[90,2] + -10.023;
   1:L PR[91] R[100]mm/sec CNT100;
   1:  PR[91,1] = PR[90,1] + 42.658;
   1:  PR[91,2] = PR[90,2] + -5.521;
   1:L PR[91] R[100]mm/sec CNT100;
   1:  PR[91,1] = PR[90,1] + 43.285;
   1:  PR[91,2] = PR[90,2] + -0.729;
   1:L PR[91] R[100]mm/sec CNT100;
   1:  PR[91,1] = PR[90,1] + 42.659;
   1:  PR[91,2] = PR[90,2] + 4.062;
   1:L PR[91] R[100]mm/sec CNT100;
   1:  PR[91,1] = PR[90,1] + 40.787;
   1:  PR[91,2] = PR[90,2] + 8.584;
   1:L PR[91] R[100]mm/sec CNT100;
   1:  PR[91,1] = PR[90,1] + 37.851;
   1:  PR[91,2] = PR[90,2] + 12.419;
   1:L PR[91] R[100]mm/sec CNT100;
   1:  PR[91,1] = PR[90,1] + 34.001;
   1:  PR[91,2] = PR[90,2] + 15.387;
   1:L PR[91] R[100]mm/sec CNT100TB   .50sec,CALL END_PUD;
   1:  PR[92] = PR[91];
   1:  PR[92,3] = PR[92,3] + 20;
   1:J PR[92] 10% FINE;
   1:  PR[91,1] = PR[90,1] + -17.097;
   1:  PR[91,2] = PR[90,2] + -17.840;
   1:  PR[92] = PR[91];
   1:  PR[92,3] = PR[92,3] + 20;
   1:J PR[92] 10% FINE;
   1:L PR[91] R[100]mm/sec CNT100;
   1:  CALL LASER_DRAHT_START;
   1:  PR[91,1] = PR[90,1] + -15.887;
   1:  PR[91,2] = PR[90,2] + -17.446;
   1:L PR[91] R[100]mm/sec CNT100;
   1:  PR[91,1] = PR[90,1] + -13.580;
   1:  PR[91,2] = PR[90,2] + -16.033;
   1:L PR[91] R[100]mm/sec CNT100;
   1:  PR[91,1] = PR[90,1] + -12.297;
   1:  PR[91,2] = PR[90,2] + -15.265;
   1:L PR[91] R[100]mm/sec CNT100;
   1:  PR[91,1] = PR[90,1] + -9.292;
   1:  PR[91,2] = PR[90,2] + -12.348;
   1:L PR[91] R[100]mm/sec CNT100;
   1:  PR[91,1] = PR[90,1] + -7.017;
   1:  PR[91,2] = PR[90,2] + -8.827;
   1:L PR[91] R[100]mm/sec CNT100;
   1:  PR[91,1] = PR[90,1] + -5.603;
   1:  PR[91,2] = PR[90,2] + -4.887;
   1:L PR[91] R[100]mm/sec CNT100;
   1:  PR[91,1] = PR[90,1] + -5.363;
   1:  PR[91,2] = PR[90,2] + -2.813;
   1:L PR[91] R[100]mm/sec CNT100;
   1:  PR[91,1] = PR[90,1] + -5.148;
   1:  PR[91,2] = PR[90,2] + -0.741;
   1:L PR[91] R[100]mm/sec CNT100;
   1:  PR[91,1] = PR[90,1] + -5.385;
   1:  PR[91,2] = PR[90,2] + 1.312;
   1:L PR[91] R[100]mm/sec CNT100;
   1:  PR[91,1] = PR[90,1] + -5.378;
   1:  PR[91,2] = PR[90,2] + 1.494;
   1:L PR[91] R[100]mm/sec CNT100;
   1:  PR[91,1] = PR[90,1] + -5.603;
   1:  PR[91,2] = PR[90,2] + 3.428;
   1:L PR[91] R[100]mm/sec CNT100;
   1:  PR[91,1] = PR[90,1] + -7.018;
   1:  PR[91,2] = PR[90,2] + 7.371;
   1:L PR[91] R[100]mm/sec CNT100;
   1:  PR[91,1] = PR[90,1] + -8.249;
   1:  PR[91,2] = PR[90,2] + 9.288;
   1:L PR[91] R[100]mm/sec CNT100;
   1:  PR[91,1] = PR[90,1] + -9.289;
   1:  PR[91,2] = PR[90,2] + 10.887;
   1:L PR[91] R[100]mm/sec CNT100;
   1:  PR[91,1] = PR[90,1] + -12.302;
   1:  PR[91,2] = PR[90,2] + 13.811;
   1:L PR[91] R[100]mm/sec CNT100;
   1:  PR[91,1] = PR[90,1] + -15.890;
   1:  PR[91,2] = PR[90,2] + 15.989;
   1:L PR[91] R[100]mm/sec CNT100;
   1:  PR[91,1] = PR[90,1] + -19.870;
   1:  PR[91,2] = PR[90,2] + 17.317;
   1:L PR[91] R[100]mm/sec CNT100;
   1:  PR[91,1] = PR[90,1] + -24.038;
   1:  PR[91,2] = PR[90,2] + 17.738;
   1:L PR[91] R[100]mm/sec CNT100;
   1:  PR[91,1] = PR[90,1] + -28.187;
   1:  PR[91,2] = PR[90,2] + 17.232;
   1:L PR[91] R[100]mm/sec CNT100;
   1:  PR[91,1] = PR[90,1] + -32.112;
   1:  PR[91,2] = PR[90,2] + 15.834;
   1:L PR[91] R[100]mm/sec CNT100;
   1:  PR[91,1] = PR[90,1] + -35.275;
   1:  PR[91,2] = PR[90,2] + 13.838;
   1:L PR[91] R[100]mm/sec CNT100;
   1:  PR[91,1] = PR[90,1] + -35.612;
   1:  PR[91,2] = PR[90,2] + 13.622;
   1:L PR[91] R[100]mm/sec CNT100;
   1:  PR[91,1] = PR[90,1] + -38.535;
   1:  PR[91,2] = PR[90,2] + 10.694;
   1:L PR[91] R[100]mm/sec CNT100;
   1:  PR[91,1] = PR[90,1] + -40.725;
   1:  PR[91,2] = PR[90,2] + 7.211;
   1:L PR[91] R[100]mm/sec CNT100;
   1:  PR[91,1] = PR[90,1] + -42.082;
   1:  PR[91,2] = PR[90,2] + 3.340;
   1:L PR[91] R[100]mm/sec CNT100;
   1:  PR[91,1] = PR[90,1] + -42.545;
   1:  PR[91,2] = PR[90,2] + -0.746;
   1:L PR[91] R[100]mm/sec CNT100;
   1:  PR[91,1] = PR[90,1] + -42.560;
   1:  PR[91,2] = PR[90,2] + -0.819;
   1:L PR[91] R[100]mm/sec CNT100;
   1:  PR[91,1] = PR[90,1] + -42.412;
   1:  PR[91,2] = PR[90,2] + -2.127;
   1:L PR[91] R[100]mm/sec CNT100;
   1:  PR[91,1] = PR[90,1] + -42.093;
   1:  PR[91,2] = PR[90,2] + -4.697;
   1:L PR[91] R[100]mm/sec CNT100;
   1:  PR[91,1] = PR[90,1] + -42.081;
   1:  PR[91,2] = PR[90,2] + -4.800;
   1:L PR[91] R[100]mm/sec CNT100;
   1:  PR[91,1] = PR[90,1] + -40.725;
   1:  PR[91,2] = PR[90,2] + -8.670;
   1:L PR[91] R[100]mm/sec CNT100;
   1:  PR[91,1] = PR[90,1] + -38.535;
   1:  PR[91,2] = PR[90,2] + -12.153;
   1:L PR[91] R[100]mm/sec CNT100;
   1:  PR[91,1] = PR[90,1] + -35.617;
   1:  PR[91,2] = PR[90,2] + -15.076;
   1:L PR[91] R[100]mm/sec CNT100;
   1:  PR[91,1] = PR[90,1] + -32.111;
   1:  PR[91,2] = PR[90,2] + -17.294;
   1:L PR[91] R[100]mm/sec CNT100;
   1:  PR[91,1] = PR[90,1] + -28.187;
   1:  PR[91,2] = PR[90,2] + -18.691;
   1:L PR[91] R[100]mm/sec CNT100;
   1:  PR[91,1] = PR[90,1] + -24.041;
   1:  PR[91,2] = PR[90,2] + -19.196;
   1:L PR[91] R[100]mm/sec CNT100;
   1:  PR[91,1] = PR[90,1] + -20.916;
   1:  PR[91,2] = PR[90,2] + -18.872;
   1:L PR[91] R[100]mm/sec CNT100;
   1:  PR[91,1] = PR[90,1] + -19.865;
   1:  PR[91,2] = PR[90,2] + -18.774;
   1:L PR[91] R[100]mm/sec CNT100;
   1:  PR[91,1] = PR[90,1] + -17.097;
   1:  PR[91,2] = PR[90,2] + -17.840;
   1:L PR[91] R[100]mm/sec CNT100TB   .50sec,CALL END_PUD;
   1:  PR[92] = PR[91];
   1:  PR[92,3] = PR[92,3] + 20;
   1:J PR[92] 10% FINE;
   1:  PR[91,1] = PR[90,1] + -54.561;
   1:  PR[91,2] = PR[90,2] + 2.063;
   1:  PR[92] = PR[91];
   1:  PR[92,3] = PR[92,3] + 20;
   1:J PR[92] 10% FINE;
   1:L PR[91] R[100]mm/sec CNT100;
   1:  CALL LASER_DRAHT_START;
   1:  PR[91,1] = PR[90,1] + -54.685;
   1:  PR[91,2] = PR[90,2] + 3.153;
   1:L PR[91] R[100]mm/sec CNT100;
   1:  PR[91,1] = PR[90,1] + -55.975;
   1:  PR[91,2] = PR[90,2] + 6.856;
   1:L PR[91] R[100]mm/sec CNT100;
   1:  PR[91,1] = PR[90,1] + -58.056;
   1:  PR[91,2] = PR[90,2] + 10.208;
   1:L PR[91] R[100]mm/sec CNT100;
   1:  PR[91,1] = PR[90,1] + -60.821;
   1:  PR[91,2] = PR[90,2] + 13.062;
   1:L PR[91] R[100]mm/sec CNT100;
   1:  PR[91,1] = PR[90,1] + -62.566;
   1:  PR[91,2] = PR[90,2] + 14.231;
   1:L PR[91] R[100]mm/sec CNT100;
   1:  PR[91,1] = PR[90,1] + -64.123;
   1:  PR[91,2] = PR[90,2] + 15.317;
   1:L PR[91] R[100]mm/sec CNT100;
   1:  PR[91,1] = PR[90,1] + -67.733;
   1:  PR[91,2] = PR[90,2] + 16.848;
   1:L PR[91] R[100]mm/sec CNT100;
   1:  PR[91,1] = PR[90,1] + -71.582;
   1:  PR[91,2] = PR[90,2] + 17.604;
   1:L PR[91] R[100]mm/sec CNT100;
   1:  PR[91,1] = PR[90,1] + -72.515;
   1:  PR[91,2] = PR[90,2] + 17.599;
   1:L PR[91] R[100]mm/sec CNT100;
   1:  PR[91,1] = PR[90,1] + -75.485;
   1:  PR[91,2] = PR[90,2] + 17.559;
   1:L PR[91] R[100]mm/sec CNT100;
   1:  PR[91,1] = PR[90,1] + -79.292;
   1:  PR[91,2] = PR[90,2] + 16.720;
   1:L PR[91] R[100]mm/sec CNT100;
   1:  PR[91,1] = PR[90,1] + -82.832;
   1:  PR[91,2] = PR[90,2] + 15.127;
   1:L PR[91] R[100]mm/sec CNT100;
   1:  PR[91,1] = PR[90,1] + -85.955;
   1:  PR[91,2] = PR[90,2] + 12.854;
   1:L PR[91] R[100]mm/sec CNT100;
   1:  PR[91,1] = PR[90,1] + -88.530;
   1:  PR[91,2] = PR[90,2] + 9.999;
   1:L PR[91] R[100]mm/sec CNT100;
   1:  PR[91,1] = PR[90,1] + -90.450;
   1:  PR[91,2] = PR[90,2] + 6.687;
   1:L PR[91] R[100]mm/sec CNT100;
   1:  PR[91,1] = PR[90,1] + -91.634;
   1:  PR[91,2] = PR[90,2] + 3.058;
   1:L PR[91] R[100]mm/sec CNT100;
   1:  PR[91,1] = PR[90,1] + -91.911;
   1:  PR[91,2] = PR[90,2] + 0.465;
   1:L PR[91] R[100]mm/sec CNT100;
   1:  PR[91,1] = PR[90,1] + -91.994;
   1:  PR[91,2] = PR[90,2] + 0.072;
   1:L PR[91] R[100]mm/sec CNT100;
   1:  PR[91,1] = PR[90,1] + -92.123;
   1:  PR[91,2] = PR[90,2] + -0.775;
   1:L PR[91] R[100]mm/sec CNT100;
   1:  PR[91,1] = PR[90,1] + -91.948;
   1:  PR[91,2] = PR[90,2] + -2.426;
   1:L PR[91] R[100]mm/sec CNT100;
   1:  PR[91,1] = PR[90,1] + -91.797;
   1:  PR[91,2] = PR[90,2] + -3.381;
   1:L PR[91] R[100]mm/sec CNT100;
   1:  PR[91,1] = PR[90,1] + -91.731;
   1:  PR[91,2] = PR[90,2] + -3.660;
   1:L PR[91] R[100]mm/sec CNT100;
   1:  PR[91,1] = PR[90,1] + -91.642;
   1:  PR[91,2] = PR[90,2] + -4.517;
   1:L PR[91] R[100]mm/sec CNT100;
   1:  PR[91,1] = PR[90,1] + -90.701;
   1:  PR[91,2] = PR[90,2] + -7.387;
   1:L PR[91] R[100]mm/sec CNT100;
   1:  PR[91,1] = PR[90,1] + -90.455;
   1:  PR[91,2] = PR[90,2] + -8.145;
   1:L PR[91] R[100]mm/sec CNT100;
   1:  PR[91,1] = PR[90,1] + -88.530;
   1:  PR[91,2] = PR[90,2] + -11.455;
   1:L PR[91] R[100]mm/sec CNT100;
   1:  PR[91,1] = PR[90,1] + -85.949;
   1:  PR[91,2] = PR[90,2] + -14.312;
   1:L PR[91] R[100]mm/sec CNT100;
   1:  PR[91,1] = PR[90,1] + -82.816;
   1:  PR[91,2] = PR[90,2] + -16.588;
   1:L PR[91] R[100]mm/sec CNT100;
   1:  PR[91,1] = PR[90,1] + -79.264;
   1:  PR[91,2] = PR[90,2] + -18.184;
   1:L PR[91] R[100]mm/sec CNT100;
   1:  PR[91,1] = PR[90,1] + -75.449;
   1:  PR[91,2] = PR[90,2] + -19.025;
   1:L PR[91] R[100]mm/sec CNT100;
   1:  PR[91,1] = PR[90,1] + -73.578;
   1:  PR[91,2] = PR[90,2] + -19.039;
   1:L PR[91] R[100]mm/sec CNT100;
   1:  PR[91,1] = PR[90,1] + -71.520;
   1:  PR[91,2] = PR[90,2] + -19.074;
   1:L PR[91] R[100]mm/sec CNT100;
   1:  PR[91,1] = PR[90,1] + -70.024;
   1:  PR[91,2] = PR[90,2] + -18.773;
   1:L PR[91] R[100]mm/sec CNT100;
   1:  PR[91,1] = PR[90,1] + -67.652;
   1:  PR[91,2] = PR[90,2] + -18.321;
   1:L PR[91] R[100]mm/sec CNT100;
   1:  PR[91,1] = PR[90,1] + -64.027;
   1:  PR[91,2] = PR[90,2] + -16.794;
   1:L PR[91] R[100]mm/sec CNT100;
   1:  PR[91,1] = PR[90,1] + -60.793;
   1:  PR[91,2] = PR[90,2] + -14.551;
   1:L PR[91] R[100]mm/sec CNT100;
   1:  PR[91,1] = PR[90,1] + -58.102;
   1:  PR[91,2] = PR[90,2] + -11.685;
   1:L PR[91] R[100]mm/sec CNT100;
   1:  PR[91,1] = PR[90,1] + -56.062;
   1:  PR[91,2] = PR[90,2] + -8.314;
   1:L PR[91] R[100]mm/sec CNT100;
   1:  PR[91,1] = PR[90,1] + -54.754;
   1:  PR[91,2] = PR[90,2] + -4.602;
   1:L PR[91] R[100]mm/sec CNT100;
   1:  PR[91,1] = PR[90,1] + -54.327;
   1:  PR[91,2] = PR[90,2] + -0.916;
   1:L PR[91] R[100]mm/sec CNT100;
   1:  PR[91,1] = PR[90,1] + -54.315;
   1:  PR[91,2] = PR[90,2] + -0.745;
   1:L PR[91] R[100]mm/sec CNT100;
   1:  PR[91,1] = PR[90,1] + -54.561;
   1:  PR[91,2] = PR[90,2] + 2.063;
   1:L PR[91] R[100]mm/sec CNT100TB   .50sec,CALL END_PUD;
   1:  PR[92] = PR[91];
   1:  PR[92,3] = PR[92,3] + 20;
   1:J PR[92] 10% FINE;
   1:  PR[91] = PR[90];
   1:  PR[91,1] = PR[90,1] + 53.000;
   1:  PR[91,2] = PR[90,2] + 3.621;
   1:  PR[91,3] = PR[90,3] + 24.895;
   1:  PR[92] = PR[91];
   1:  PR[92,3] = PR[92,3] + 20;
   1:J PR[92] 10% FINE;
   1:L PR[91] R[100]mm/sec CNT100;
   1:  CALL LASER_DRAHT_START;
   1:  PR[91,1] = PR[90,1] + 52.821;
   1:  PR[91,2] = PR[90,2] + 2.212;
   1:L PR[91] R[100]mm/sec CNT100;
   1:  PR[91,1] = PR[90,1] + 52.724;
   1:  PR[91,2] = PR[90,2] + 0.636;
   1:L PR[91] R[100]mm/sec CNT100;
   1:  PR[91,1] = PR[90,1] + 52.542;
   1:  PR[91,2] = PR[90,2] + -0.787;
   1:L PR[91] R[100]mm/sec CNT100;
   1:  PR[91,1] = PR[90,1] + 52.637;
   1:  PR[91,2] = PR[90,2] + -2.151;
   1:L PR[91] R[100]mm/sec CNT100;
   1:  PR[91,1] = PR[90,1] + 53.002;
   1:  PR[91,2] = PR[90,2] + -5.092;
   1:L PR[91] R[100]mm/sec CNT100;
   1:  PR[91,1] = PR[90,1] + 53.615;
   1:  PR[91,2] = PR[90,2] + -6.680;
   1:L PR[91] R[100]mm/sec CNT100;
   1:  PR[91,1] = PR[90,1] + 54.608;
   1:  PR[91,2] = PR[90,2] + -9.191;
   1:L PR[91] R[100]mm/sec CNT100;
   1:  PR[91,1] = PR[90,1] + 55.896;
   1:  PR[91,2] = PR[90,2] + -11.041;
   1:L PR[91] R[100]mm/sec CNT100;
   1:  PR[91,1] = PR[90,1] + 57.163;
   1:  PR[91,2] = PR[90,2] + -12.813;
   1:L PR[91] R[100]mm/sec CNT100;
   1:  PR[91,1] = PR[90,1] + 59.431;
   1:  PR[91,2] = PR[90,2] + -14.842;
   1:L PR[91] R[100]mm/sec CNT100;
   1:  PR[91,1] = PR[90,1] + 60.497;
   1:  PR[91,2] = PR[90,2] + -15.768;
   1:L PR[91] R[100]mm/sec CNT100;
   1:  PR[91,1] = PR[90,1] + 64.431;
   1:  PR[91,2] = PR[90,2] + -17.929;
   1:L PR[91] R[100]mm/sec CNT100;
   1:  PR[91,1] = PR[90,1] + 68.003;
   1:  PR[91,2] = PR[90,2] + -18.978;
   1:L PR[91] R[100]mm/sec CNT100;
   1:  PR[91,1] = PR[90,1] + 68.730;
   1:  PR[91,2] = PR[90,2] + -19.208;
   1:L PR[91] R[100]mm/sec CNT100;
   1:  PR[91,1] = PR[90,1] + 73.036;
   1:  PR[91,2] = PR[90,2] + -19.579;
   1:L PR[91] R[100]mm/sec CNT100;
   1:  PR[91,1] = PR[90,1] + 73.551;
   1:  PR[91,2] = PR[90,2] + -19.516;
   1:L PR[91] R[100]mm/sec CNT100;
   1:  PR[91,1] = PR[90,1] + 77.283;
   1:  PR[91,2] = PR[90,2] + -19.011;
   1:L PR[91] R[100]mm/sec CNT100;
   1:  PR[91,1] = PR[90,1] + 78.268;
   1:  PR[91,2] = PR[90,2] + -18.660;
   1:L PR[91] R[100]mm/sec CNT100;
   1:  PR[91,1] = PR[90,1] + 81.280;
   1:  PR[91,2] = PR[90,2] + -17.550;
   1:L PR[91] R[100]mm/sec CNT100;
   1:  PR[91,1] = PR[90,1] + 82.526;
   1:  PR[91,2] = PR[90,2] + -16.763;
   1:L PR[91] R[100]mm/sec CNT100;
   1:  PR[91,1] = PR[90,1] + 84.834;
   1:  PR[91,2] = PR[90,2] + -15.274;
   1:L PR[91] R[100]mm/sec CNT100;
   1:  PR[91,1] = PR[90,1] + 87.792;
   1:  PR[91,2] = PR[90,2] + -12.292;
   1:L PR[91] R[100]mm/sec CNT100;
   1:  PR[91,1] = PR[90,1] + 90.007;
   1:  PR[91,2] = PR[90,2] + -8.757;
   1:L PR[91] R[100]mm/sec CNT100;
   1:  PR[91,1] = PR[90,1] + 90.734;
   1:  PR[91,2] = PR[90,2] + -6.688;
   1:L PR[91] R[100]mm/sec CNT100;
   1:  PR[91,1] = PR[90,1] + 91.375;
   1:  PR[91,2] = PR[90,2] + -4.842;
   1:L PR[91] R[100]mm/sec CNT100;
   1:  PR[91,1] = PR[90,1] + 91.645;
   1:  PR[91,2] = PR[90,2] + -2.502;
   1:L PR[91] R[100]mm/sec CNT100;
   1:  PR[91,1] = PR[90,1] + 91.921;
   1:  PR[91,2] = PR[90,2] + -0.692;
   1:L PR[91] R[100]mm/sec CNT100;
   1:  PR[91,1] = PR[90,1] + 91.811;
   1:  PR[91,2] = PR[90,2] + 0.265;
   1:L PR[91] R[100]mm/sec CNT100;
   1:  PR[91,1] = PR[90,1] + 91.584;
   1:  PR[91,2] = PR[90,2] + 1.492;
   1:L PR[91] R[100]mm/sec CNT100;
   1:  PR[91,1] = PR[90,1] + 91.374;
   1:  PR[91,2] = PR[90,2] + 3.385;
   1:L PR[91] R[100]mm/sec CNT100;
   1:  PR[91,1] = PR[90,1] + 90.006;
   1:  PR[91,2] = PR[90,2] + 7.300;
   1:L PR[91] R[100]mm/sec CNT100;
   1:  PR[91,1] = PR[90,1] + 87.795;
   1:  PR[91,2] = PR[90,2] + 10.829;
   1:L PR[91] R[100]mm/sec CNT100;
   1:  PR[91,1] = PR[90,1] + 86.441;
   1:  PR[91,2] = PR[90,2] + 12.181;
   1:L PR[91] R[100]mm/sec CNT100;
   1:  PR[91,1] = PR[90,1] + 84.838;
   1:  PR[91,2] = PR[90,2] + 13.810;
   1:L PR[91] R[100]mm/sec CNT100;
   1:  PR[91,1] = PR[90,1] + 83.443;
   1:  PR[91,2] = PR[90,2] + 14.690;
   1:L PR[91] R[100]mm/sec CNT100;
   1:  PR[91,1] = PR[90,1] + 81.280;
   1:  PR[91,2] = PR[90,2] + 16.088;
   1:L PR[91] R[100]mm/sec CNT100;
   1:  PR[91,1] = PR[90,1] + 80.040;
   1:  PR[91,2] = PR[90,2] + 16.529;
   1:L PR[91] R[100]mm/sec CNT100;
   1:  PR[91,1] = PR[90,1] + 77.283;
   1:  PR[91,2] = PR[90,2] + 17.549;
   1:L PR[91] R[100]mm/sec CNT100;
   1:  PR[91,1] = PR[90,1] + 76.379;
   1:  PR[91,2] = PR[90,2] + 17.659;
   1:L PR[91] R[100]mm/sec CNT100;
   1:  PR[91,1] = PR[90,1] + 73.023;
   1:  PR[91,2] = PR[90,2] + 18.119;
   1:L PR[91] R[100]mm/sec CNT100;
   1:  PR[91,1] = PR[90,1] + 68.730;
   1:  PR[91,2] = PR[90,2] + 17.749;
   1:L PR[91] R[100]mm/sec CNT100;
   1:  PR[91,1] = PR[90,1] + 68.004;
   1:  PR[91,2] = PR[90,2] + 17.519;
   1:L PR[91] R[100]mm/sec CNT100;
   1:  PR[91,1] = PR[90,1] + 64.435;
   1:  PR[91,2] = PR[90,2] + 16.472;
   1:L PR[91] R[100]mm/sec CNT100;
   1:  PR[91,1] = PR[90,1] + 61.289;
   1:  PR[91,2] = PR[90,2] + 14.723;
   1:L PR[91] R[100]mm/sec CNT100;
   1:  PR[91,1] = PR[90,1] + 60.499;
   1:  PR[91,2] = PR[90,2] + 14.306;
   1:L PR[91] R[100]mm/sec CNT100;
   1:  PR[91,1] = PR[90,1] + 58.310;
   1:  PR[91,2] = PR[90,2] + 12.338;
   1:L PR[91] R[100]mm/sec CNT100;
   1:  PR[91,1] = PR[90,1] + 57.164;
   1:  PR[91,2] = PR[90,2] + 11.349;
   1:L PR[91] R[100]mm/sec CNT100;
   1:  PR[91,1] = PR[90,1] + 55.827;
   1:  PR[91,2] = PR[90,2] + 9.423;
   1:L PR[91] R[100]mm/sec CNT100;
   1:  PR[91,1] = PR[90,1] + 54.608;
   1:  PR[91,2] = PR[90,2] + 7.726;
   1:L PR[91] R[100]mm/sec CNT100;
   1:  PR[91,1] = PR[90,1] + 53.945;
   1:  PR[91,2] = PR[90,2] + 6.004;
   1:L PR[91] R[100]mm/sec CNT100;
   1:  PR[91,1] = PR[90,1] + 53.000;
   1:  PR[91,2] = PR[90,2] + 3.621;
   1:L PR[91] R[100]mm/sec CNT100TB   .50sec,CALL END_PUD;
   1:  PR[92] = PR[91];
   1:  PR[92,3] = PR[92,3] + 20;
   1:J PR[92] 10% FINE;
   1:  PR[91,1] = PR[90,1] + 8.268;
   1:  PR[91,2] = PR[90,2] + 8.694;
   1:  PR[92] = PR[91];
   1:  PR[92,3] = PR[92,3] + 20;
   1:J PR[92] 10% FINE;
   1:L PR[91] R[100]mm/sec CNT100;
   1:  CALL LASER_DRAHT_START;
   1:  PR[91,1] = PR[90,1] + 6.376;
   1:  PR[91,2] = PR[90,2] + 4.150;
   1:L PR[91] R[100]mm/sec CNT100;
   1:  PR[91,1] = PR[90,1] + 5.730;
   1:  PR[91,2] = PR[90,2] + -0.729;
   1:L PR[91] R[100]mm/sec CNT100;
   1:  PR[91,1] = PR[90,1] + 6.377;
   1:  PR[91,2] = PR[90,2] + -5.610;
   1:L PR[91] R[100]mm/sec CNT100;
   1:  PR[91,1] = PR[90,1] + 8.269;
   1:  PR[91,2] = PR[90,2] + -10.154;
   1:L PR[91] R[100]mm/sec CNT100;
   1:  PR[91,1] = PR[90,1] + 11.275;
   1:  PR[91,2] = PR[90,2] + -14.051;
   1:L PR[91] R[100]mm/sec CNT100;
   1:  PR[91,1] = PR[90,1] + 15.188;
   1:  PR[91,2] = PR[90,2] + -17.031;
   1:L PR[91] R[100]mm/sec CNT100;
   1:  PR[91,1] = PR[90,1] + 19.740;
   1:  PR[91,2] = PR[90,2] + -18.897;
   1:L PR[91] R[100]mm/sec CNT100;
   1:  PR[91,1] = PR[90,1] + 20.215;
   1:  PR[91,2] = PR[90,2] + -18.959;
   1:L PR[91] R[100]mm/sec CNT100;
   1:  PR[91,1] = PR[90,1] + 24.608;
   1:  PR[91,2] = PR[90,2] + -19.520;
   1:L PR[91] R[100]mm/sec CNT100;
   1:  PR[91,1] = PR[90,1] + 29.471;
   1:  PR[91,2] = PR[90,2] + -18.863;
   1:L PR[91] R[100]mm/sec CNT100;
   1:  PR[91,1] = PR[90,1] + 34.002;
   1:  PR[91,2] = PR[90,2] + -16.973;
   1:L PR[91] R[100]mm/sec CNT100;
   1:  PR[91,1] = PR[90,1] + 34.223;
   1:  PR[91,2] = PR[90,2] + -16.805;
   1:L PR[91] R[100]mm/sec CNT100;
   1:  PR[91,1] = PR[90,1] + 37.872;
   1:  PR[91,2] = PR[90,2] + -13.991;
   1:L PR[91] R[100]mm/sec CNT100;
   1:  PR[91,1] = PR[90,1] + 40.847;
   1:  PR[91,2] = PR[90,2] + -10.106;
   1:L PR[91] R[100]mm/sec CNT100;
   1:  PR[91,1] = PR[90,1] + 42.712;
   1:  PR[91,2] = PR[90,2] + -5.626;
   1:L PR[91] R[100]mm/sec CNT100;
   1:  PR[91,1] = PR[90,1] + 42.747;
   1:  PR[91,2] = PR[90,2] + -5.491;
   1:L PR[91] R[100]mm/sec CNT100;
   1:  PR[91,1] = PR[90,1] + 43.338;
   1:  PR[91,2] = PR[90,2] + -0.994;
   1:L PR[91] R[100]mm/sec CNT100;
   1:  PR[91,1] = PR[90,1] + 43.358;
   1:  PR[91,2] = PR[90,2] + -0.772;
   1:L PR[91] R[100]mm/sec CNT100;
   1:  PR[91,1] = PR[90,1] + 42.777;
   1:  PR[91,2] = PR[90,2] + 3.645;
   1:L PR[91] R[100]mm/sec CNT100;
   1:  PR[91,1] = PR[90,1] + 42.740;
   1:  PR[91,2] = PR[90,2] + 4.053;
   1:L PR[91] R[100]mm/sec CNT100;
   1:  PR[91,1] = PR[90,1] + 42.704;
   1:  PR[91,2] = PR[90,2] + 4.191;
   1:L PR[91] R[100]mm/sec CNT100;
   1:  PR[91,1] = PR[90,1] + 40.933;
   1:  PR[91,2] = PR[90,2] + 8.481;
   1:L PR[91] R[100]mm/sec CNT100;
   1:  PR[91,1] = PR[90,1] + 40.872;
   1:  PR[91,2] = PR[90,2] + 8.614;
   1:L PR[91] R[100]mm/sec CNT100;
   1:  PR[91,1] = PR[90,1] + 37.870;
   1:  PR[91,2] = PR[90,2] + 12.534;
   1:L PR[91] R[100]mm/sec CNT100;
   1:  PR[91,1] = PR[90,1] + 33.990;
   1:  PR[91,2] = PR[90,2] + 15.520;
   1:L PR[91] R[100]mm/sec CNT100;
   1:  PR[91,1] = PR[90,1] + 29.789;
   1:  PR[91,2] = PR[90,2] + 17.276;
   1:L PR[91] R[100]mm/sec CNT100;
   1:  PR[91,1] = PR[90,1] + 29.476;
   1:  PR[91,2] = PR[90,2] + 17.404;
   1:L PR[91] R[100]mm/sec CNT100;
   1:  PR[91,1] = PR[90,1] + 24.605;
   1:  PR[91,2] = PR[90,2] + 18.061;
   1:L PR[91] R[100]mm/sec CNT100;
   1:  PR[91,1] = PR[90,1] + 19.733;
   1:  PR[91,2] = PR[90,2] + 17.436;
   1:L PR[91] R[100]mm/sec CNT100;
   1:  PR[91,1] = PR[90,1] + 15.692;
   1:  PR[91,2] = PR[90,2] + 15.781;
   1:L PR[91] R[100]mm/sec CNT100;
   1:  PR[91,1] = PR[90,1] + 15.188;
   1:  PR[91,2] = PR[90,2] + 15.573;
   1:L PR[91] R[100]mm/sec CNT100;
   1:  PR[91,1] = PR[90,1] + 11.273;
   1:  PR[91,2] = PR[90,2] + 12.590;
   1:L PR[91] R[100]mm/sec CNT100;
   1:  PR[91,1] = PR[90,1] + 8.268;
   1:  PR[91,2] = PR[90,2] + 8.694;
   1:L PR[91] R[100]mm/sec CNT100TB   .50sec,CALL END_PUD;
   1:  PR[92] = PR[91];
   1:  PR[92,3] = PR[92,3] + 20;
   1:J PR[92] 10% FINE;
   1:  PR[91,1] = PR[90,1] + -28.012;
   1:  PR[91,2] = PR[90,2] + 17.312;
   1:  PR[92] = PR[91];
   1:  PR[92,3] = PR[92,3] + 20;
   1:J PR[92] 10% FINE;
   1:L PR[91] R[100]mm/sec CNT100;
   1:  CALL LASER_DRAHT_START;
   1:  PR[91,1] = PR[90,1] + -31.954;
   1:  PR[91,2] = PR[90,2] + 15.904;
   1:L PR[91] R[100]mm/sec CNT100;
   1:  PR[91,1] = PR[90,1] + -34.716;
   1:  PR[91,2] = PR[90,2] + 14.161;
   1:L PR[91] R[100]mm/sec CNT100;
   1:  PR[91,1] = PR[90,1] + -35.466;
   1:  PR[91,2] = PR[90,2] + 13.679;
   1:L PR[91] R[100]mm/sec CNT100;
   1:  PR[91,1] = PR[90,1] + -38.398;
   1:  PR[91,2] = PR[90,2] + 10.738;
   1:L PR[91] R[100]mm/sec CNT100;
   1:  PR[91,1] = PR[90,1] + -40.595;
   1:  PR[91,2] = PR[90,2] + 7.241;
   1:L PR[91] R[100]mm/sec CNT100;
   1:  PR[91,1] = PR[90,1] + -41.956;
   1:  PR[91,2] = PR[90,2] + 3.355;
   1:L PR[91] R[100]mm/sec CNT100;
   1:  PR[91,1] = PR[90,1] + -42.372;
   1:  PR[91,2] = PR[90,2] + -0.312;
   1:L PR[91] R[100]mm/sec CNT100;
   1:  PR[91,1] = PR[90,1] + -42.457;
   1:  PR[91,2] = PR[90,2] + -0.729;
   1:L PR[91] R[100]mm/sec CNT100;
   1:  PR[91,1] = PR[90,1] + -42.014;
   1:  PR[91,2] = PR[90,2] + -4.284;
   1:L PR[91] R[100]mm/sec CNT100;
   1:  PR[91,1] = PR[90,1] + -41.955;
   1:  PR[91,2] = PR[90,2] + -4.815;
   1:L PR[91] R[100]mm/sec CNT100;
   1:  PR[91,1] = PR[90,1] + -40.595;
   1:  PR[91,2] = PR[90,2] + -8.700;
   1:L PR[91] R[100]mm/sec CNT100;
   1:  PR[91,1] = PR[90,1] + -38.398;
   1:  PR[91,2] = PR[90,2] + -12.197;
   1:L PR[91] R[100]mm/sec CNT100;
   1:  PR[91,1] = PR[90,1] + -35.470;
   1:  PR[91,2] = PR[90,2] + -15.134;
   1:L PR[91] R[100]mm/sec CNT100;
   1:  PR[91,1] = PR[90,1] + -31.952;
   1:  PR[91,2] = PR[90,2] + -17.363;
   1:L PR[91] R[100]mm/sec CNT100;
   1:  PR[91,1] = PR[90,1] + -28.016;
   1:  PR[91,2] = PR[90,2] + -18.769;
   1:L PR[91] R[100]mm/sec CNT100;
   1:  PR[91,1] = PR[90,1] + -25.155;
   1:  PR[91,2] = PR[90,2] + -19.111;
   1:L PR[91] R[100]mm/sec CNT100;
   1:  PR[91,1] = PR[90,1] + -23.842;
   1:  PR[91,2] = PR[90,2] + -19.282;
   1:L PR[91] R[100]mm/sec CNT100;
   1:  PR[91,1] = PR[90,1] + -21.201;
   1:  PR[91,2] = PR[90,2] + -19.008;
   1:L PR[91] R[100]mm/sec CNT100;
   1:  PR[91,1] = PR[90,1] + -19.654;
   1:  PR[91,2] = PR[90,2] + -18.864;
   1:L PR[91] R[100]mm/sec CNT100;
   1:  PR[91,1] = PR[90,1] + -17.358;
   1:  PR[91,2] = PR[90,2] + -18.089;
   1:L PR[91] R[100]mm/sec CNT100;
   1:  PR[91,1] = PR[90,1] + -15.653;
   1:  PR[91,2] = PR[90,2] + -17.534;
   1:L PR[91] R[100]mm/sec CNT100;
   1:  PR[91,1] = PR[90,1] + -13.789;
   1:  PR[91,2] = PR[90,2] + -16.393;
   1:L PR[91] R[100]mm/sec CNT100;
   1:  PR[91,1] = PR[90,1] + -12.044;
   1:  PR[91,2] = PR[90,2] + -15.348;
   1:L PR[91] R[100]mm/sec CNT100;
   1:  PR[91,1] = PR[90,1] + -10.644;
   1:  PR[91,2] = PR[90,2] + -13.979;
   1:L PR[91] R[100]mm/sec CNT100;
   1:  PR[91,1] = PR[90,1] + -9.012;
   1:  PR[91,2] = PR[90,2] + -12.411;
   1:L PR[91] R[100]mm/sec CNT100;
   1:  PR[91,1] = PR[90,1] + -6.723;
   1:  PR[91,2] = PR[90,2] + -8.875;
   1:L PR[91] R[100]mm/sec CNT100;
   1:  PR[91,1] = PR[90,1] + -5.298;
   1:  PR[91,2] = PR[90,2] + -4.912;
   1:L PR[91] R[100]mm/sec CNT100;
   1:  PR[91,1] = PR[90,1] + -5.127;
   1:  PR[91,2] = PR[90,2] + -3.428;
   1:L PR[91] R[100]mm/sec CNT100;
   1:  PR[91,1] = PR[90,1] + -4.848;
   1:  PR[91,2] = PR[90,2] + -0.741;
   1:L PR[91] R[100]mm/sec CNT100;
   1:  PR[91,1] = PR[90,1] + -5.010;
   1:  PR[91,2] = PR[90,2] + 0.662;
   1:L PR[91] R[100]mm/sec CNT100;
   1:  PR[91,1] = PR[90,1] + -5.001;
   1:  PR[91,2] = PR[90,2] + 0.893;
   1:L PR[91] R[100]mm/sec CNT100;
   1:  PR[91,1] = PR[90,1] + -5.298;
   1:  PR[91,2] = PR[90,2] + 3.453;
   1:L PR[91] R[100]mm/sec CNT100;
   1:  PR[91,1] = PR[90,1] + -6.723;
   1:  PR[91,2] = PR[90,2] + 7.416;
   1:L PR[91] R[100]mm/sec CNT100;
   1:  PR[91,1] = PR[90,1] + -9.014;
   1:  PR[91,2] = PR[90,2] + 10.955;
   1:L PR[91] R[100]mm/sec CNT100;
   1:  PR[91,1] = PR[90,1] + -12.047;
   1:  PR[91,2] = PR[90,2] + 13.894;
   1:L PR[91] R[100]mm/sec CNT100;
   1:  PR[91,1] = PR[90,1] + -13.845;
   1:  PR[91,2] = PR[90,2] + 14.994;
   1:L PR[91] R[100]mm/sec CNT100;
   1:  PR[91,1] = PR[90,1] + -15.653;
   1:  PR[91,2] = PR[90,2] + 16.077;
   1:L PR[91] R[100]mm/sec CNT100;
   1:  PR[91,1] = PR[90,1] + -17.900;
   1:  PR[91,2] = PR[90,2] + 16.835;
   1:L PR[91] R[100]mm/sec CNT100;
   1:  PR[91,1] = PR[90,1] + -19.654;
   1:  PR[91,2] = PR[90,2] + 17.407;
   1:L PR[91] R[100]mm/sec CNT100;
   1:  PR[91,1] = PR[90,1] + -22.274;
   1:  PR[91,2] = PR[90,2] + 17.678;
   1:L PR[91] R[100]mm/sec CNT100;
   1:  PR[91,1] = PR[90,1] + -23.839;
   1:  PR[91,2] = PR[90,2] + 17.825;
   1:L PR[91] R[100]mm/sec CNT100;
   1:  PR[91,1] = PR[90,1] + -28.012;
   1:  PR[91,2] = PR[90,2] + 17.312;
   1:L PR[91] R[100]mm/sec CNT100TB   .50sec,CALL END_PUD;
   1:  PR[92] = PR[91];
   1:  PR[92,3] = PR[92,3] + 20;
   1:J PR[92] 10% FINE;
   1:  PR[91,1] = PR[90,1] + -91.965;
   1:  PR[91,2] = PR[90,2] + -0.775;
   1:  PR[92] = PR[91];
   1:  PR[92,3] = PR[92,3] + 20;
   1:J PR[92] 10% FINE;
   1:L PR[91] R[100]mm/sec CNT100;
   1:  CALL LASER_DRAHT_START;
   1:  PR[91,1] = PR[90,1] + -91.902;
   1:  PR[91,2] = PR[90,2] + -1.365;
   1:L PR[91] R[100]mm/sec CNT100;
   1:  PR[91,1] = PR[90,1] + -91.671;
   1:  PR[91,2] = PR[90,2] + -2.832;
   1:L PR[91] R[100]mm/sec CNT100;
   1:  PR[91,1] = PR[90,1] + -91.580;
   1:  PR[91,2] = PR[90,2] + -3.221;
   1:L PR[91] R[100]mm/sec CNT100;
   1:  PR[91,1] = PR[90,1] + -91.443;
   1:  PR[91,2] = PR[90,2] + -4.526;
   1:L PR[91] R[100]mm/sec CNT100;
   1:  PR[91,1] = PR[90,1] + -90.641;
   1:  PR[91,2] = PR[90,2] + -6.975;
   1:L PR[91] R[100]mm/sec CNT100;
   1:  PR[91,1] = PR[90,1] + -90.254;
   1:  PR[91,2] = PR[90,2] + -8.164;
   1:L PR[91] R[100]mm/sec CNT100;
   1:  PR[91,1] = PR[90,1] + -88.326;
   1:  PR[91,2] = PR[90,2] + -11.484;
   1:L PR[91] R[100]mm/sec CNT100;
   1:  PR[91,1] = PR[90,1] + -85.739;
   1:  PR[91,2] = PR[90,2] + -14.350;
   1:L PR[91] R[100]mm/sec CNT100;
   1:  PR[91,1] = PR[90,1] + -82.599;
   1:  PR[91,2] = PR[90,2] + -16.635;
   1:L PR[91] R[100]mm/sec CNT100;
   1:  PR[91,1] = PR[90,1] + -79.038;
   1:  PR[91,2] = PR[90,2] + -18.239;
   1:L PR[91] R[100]mm/sec CNT100;
   1:  PR[91,1] = PR[90,1] + -75.212;
   1:  PR[91,2] = PR[90,2] + -19.088;
   1:L PR[91] R[100]mm/sec CNT100;
   1:  PR[91,1] = PR[90,1] + -73.873;
   1:  PR[91,2] = PR[90,2] + -19.097;
   1:L PR[91] R[100]mm/sec CNT100;
   1:  PR[91,1] = PR[90,1] + -71.262;
   1:  PR[91,2] = PR[90,2] + -19.142;
   1:L PR[91] R[100]mm/sec CNT100;
   1:  PR[91,1] = PR[90,1] + -67.387;
   1:  PR[91,2] = PR[90,2] + -18.392;
   1:L PR[91] R[100]mm/sec CNT100;
   1:  PR[91,1] = PR[90,1] + -63.742;
   1:  PR[91,2] = PR[90,2] + -16.862;
   1:L PR[91] R[100]mm/sec CNT100;
   1:  PR[91,1] = PR[90,1] + -60.834;
   1:  PR[91,2] = PR[90,2] + -14.852;
   1:L PR[91] R[100]mm/sec CNT100;
   1:  PR[91,1] = PR[90,1] + -60.435;
   1:  PR[91,2] = PR[90,2] + -14.589;
   1:L PR[91] R[100]mm/sec CNT100;
   1:  PR[91,1] = PR[90,1] + -57.617;
   1:  PR[91,2] = PR[90,2] + -11.727;
   1:L PR[91] R[100]mm/sec CNT100;
   1:  PR[91,1] = PR[90,1] + -55.494;
   1:  PR[91,2] = PR[90,2] + -8.359;
   1:L PR[91] R[100]mm/sec CNT100;
   1:  PR[91,1] = PR[90,1] + -54.176;
   1:  PR[91,2] = PR[90,2] + -4.634;
   1:L PR[91] R[100]mm/sec CNT100;
   1:  PR[91,1] = PR[90,1] + -53.844;
   1:  PR[91,2] = PR[90,2] + -1.761;
   1:L PR[91] R[100]mm/sec CNT100;
   1:  PR[91,1] = PR[90,1] + -53.770;
   1:  PR[91,2] = PR[90,2] + -0.745;
   1:L PR[91] R[100]mm/sec CNT100;
   1:  PR[91,1] = PR[90,1] + -53.934;
   1:  PR[91,2] = PR[90,2] + 1.126;
   1:L PR[91] R[100]mm/sec CNT100;
   1:  PR[91,1] = PR[90,1] + -54.167;
   1:  PR[91,2] = PR[90,2] + 3.182;
   1:L PR[91] R[100]mm/sec CNT100;
   1:  PR[91,1] = PR[90,1] + -55.471;
   1:  PR[91,2] = PR[90,2] + 6.911;
   1:L PR[91] R[100]mm/sec CNT100;
   1:  PR[91,1] = PR[90,1] + -57.572;
   1:  PR[91,2] = PR[90,2] + 10.284;
   1:L PR[91] R[100]mm/sec CNT100;
   1:  PR[91,1] = PR[90,1] + -60.362;
   1:  PR[91,2] = PR[90,2] + 13.153;
   1:L PR[91] R[100]mm/sec CNT100;
   1:  PR[91,1] = PR[90,1] + -63.710;
   1:  PR[91,2] = PR[90,2] + 15.390;
   1:L PR[91] R[100]mm/sec CNT100;
   1:  PR[91,1] = PR[90,1] + -67.467;
   1:  PR[91,2] = PR[90,2] + 16.910;
   1:L PR[91] R[100]mm/sec CNT100;
   1:  PR[91,1] = PR[90,1] + -71.350;
   1:  PR[91,2] = PR[90,2] + 17.665;
   1:L PR[91] R[100]mm/sec CNT100;
   1:  PR[91,1] = PR[90,1] + -75.273;
   1:  PR[91,2] = PR[90,2] + 17.615;
   1:L PR[91] R[100]mm/sec CNT100;
   1:  PR[91,1] = PR[90,1] + -79.090;
   1:  PR[91,2] = PR[90,2] + 16.770;
   1:L PR[91] R[100]mm/sec CNT100;
   1:  PR[91,1] = PR[90,1] + -82.637;
   1:  PR[91,2] = PR[90,2] + 15.170;
   1:L PR[91] R[100]mm/sec CNT100;
   1:  PR[91,1] = PR[90,1] + -85.767;
   1:  PR[91,2] = PR[90,2] + 12.888;
   1:L PR[91] R[100]mm/sec CNT100;
   1:  PR[91,1] = PR[90,1] + -88.347;
   1:  PR[91,2] = PR[90,2] + 10.025;
   1:L PR[91] R[100]mm/sec CNT100;
   1:  PR[91,1] = PR[90,1] + -90.271;
   1:  PR[91,2] = PR[90,2] + 6.704;
   1:L PR[91] R[100]mm/sec CNT100;
   1:  PR[91,1] = PR[90,1] + -91.456;
   1:  PR[91,2] = PR[90,2] + 3.067;
   1:L PR[91] R[100]mm/sec CNT100;
   1:  PR[91,1] = PR[90,1] + -91.680;
   1:  PR[91,2] = PR[90,2] + 0.971;
   1:L PR[91] R[100]mm/sec CNT100;
   1:  PR[91,1] = PR[90,1] + -91.750;
   1:  PR[91,2] = PR[90,2] + 0.643;
   1:L PR[91] R[100]mm/sec CNT100;
   1:  PR[91,1] = PR[90,1] + -91.965;
   1:  PR[91,2] = PR[90,2] + -0.775;
   1:L PR[91] R[100]mm/sec CNT100TB   .50sec,CALL END_PUD;
   1:  PR[92] = PR[91];
   1:  PR[92,3] = PR[92,3] + 20;
   1:J PR[92] 10% FINE;
